LIN {X 0,Y 139.124,Z 614.225,A -85,B 0,C 180,E1 -24904.524,E2 -24904.524} C_VEL
LIN {X 0,Y 138.778,Z 622.355,A -85,B 0,C 180,E1 -24907.678,E2 -24907.678} C_VEL
LIN {X 0,Y 138.183,Z 627.369,A -85,B 0,C 180,E1 -24909.922,E2 -24909.922} C_VEL
LIN {X 0,Y 136.601,Z 635.445,A -85,B 0,C 180,E1 -24914.33,E2 -24914.33} C_VEL
LIN {X 0,Y 136.009,Z 642.268,A -85,B 0,C 180,E1 -24919.047,E2 -24919.047} C_VEL
LIN {X 0,Y 136.236,Z 647.891,A -85,B 0,C 180,E1 -24924.078,E2 -24924.078} C_VEL
LIN {X 0,Y 136.959,Z 651.569,A -85,B 0,C 180,E1 -24928.53,E2 -24928.53} C_VEL
LIN {X 0,Y 137.272,Z 652.511,A -85,B 0,C 180,E1 -24930,E2 -24930} C_VEL
LIN {X 0,Y 136.446,Z 653.751,A -85,B 0,C 180,E1 -24932.953,E2 -24932.953} C_VEL
LIN {X 0,Y 135.241,Z 654.945,A -85,B 0,C 180,E1 -24939.122,E2 -24939.122} C_VEL
LIN {X 0,Y 135.535,Z 654.719,A -85,B 0,C 180,E1 -24945.027,E2 -24945.027} C_VEL
LIN {X 0,Y 137.465,Z 653.171,A -85,B 0,C 180,E1 -24950.971,E2 -24950.971} C_VEL
LIN {X 0,Y 141.156,Z 650.311,A -85,B 0,C 180,E1 -24956.622,E2 -24956.622} C_VEL
LIN {X 0,Y 146.54,Z 646.045,A -85,B 0,C 180,E1 -24961.841,E2 -24961.841} C_VEL
LIN {X 0,Y 151.131,Z 641.889,A -85,B 0,C 180,E1 -24965.542,E2 -24965.542} C_VEL
LIN {X 0,Y 157.922,Z 634.932,A -85,B 0,C 180,E1 -24970.188,E2 -24970.188} C_VEL
LIN {X 0,Y 163.15,Z 628.696,A -85,B 0,C 180,E1 -24973.57,E2 -24973.57} C_VEL
LIN {X 0,Y 169.127,Z 620.28,A -85,B 0,C 180,E1 -24977.528,E2 -24977.528} C_VEL
LIN {X 0,Y 174.471,Z 611.295,A -85,B 0,C 180,E1 -24981.463,E2 -24981.463} C_VEL
LIN {X 0,Y 175.351,Z 609.732,A -85,B 0,C 180,E1 -24982.142,E2 -24982.142} C_VEL
LIN {X 0,Y 176.005,Z 607.9,A -85,B 0,C 180,E1 -24983.205,E2 -24983.205} C_VEL
LIN {X 0,Y 176.463,Z 604.236,A -85,B 0,C 180,E1 -24986.112,E2 -24986.112} C_VEL
LIN {X 0,Y 176.98,Z 601.228,A -85,B 0,C 180,E1 -24988.92,E2 -24988.92} C_VEL
LIN {X 0,Y 177.146,Z 597.841,A -85,B 0,C 180,E1 -24994.126,E2 -24994.126} C_VEL
LIN {X 0,Y 177.528,Z 596.674,A -85,B 0,C 180,E1 -24996.68,E2 -24996.68} C_VEL
LIN {X 0,Y 177.92,Z 595.956,A -85,B 0,C 180,E1 -24999.176,E2 -24999.176} C_VEL
LIN {X 0,Y 178.33,Z 595.956,A -85,B 0,C 180,E1 -25002.881,E2 -25002.881} C_VEL
LIN {X 0,Y 178.144,Z 596.469,A -85,B 0,C 180,E1 -25004.127,E2 -25004.127} C_VEL
LIN {X 0,Y 176.937,Z 598.219,A -85,B 0,C 180,E1 -25005.914,E2 -25005.914} C_VEL
LIN {X 0,Y 173.626,Z 602.149,A -85,B 0,C 180,E1 -25008.757,E2 -25008.757} C_VEL
LIN {X 0,Y 170.434,Z 605.82,A -85,B 0,C 180,E1 -25011.758,E2 -25011.758} C_VEL
LIN {X 0,Y 170.01,Z 606.402,A -85,B 0,C 180,E1 -25012.401,E2 -25012.401} C_VEL
LIN {X 0,Y 168.927,Z 607.829,A -85,B 0,C 180,E1 -25014.03,E2 -25014.03} C_VEL
LIN {X 0,Y 161.536,Z 613.41,A -85,B 0,C 180,E1 -25017.507,E2 -25017.507} C_VEL
LIN {X 0,Y 154.657,Z 617.635,A -85,B 0,C 180,E1 -25021.293,E2 -25021.293} C_VEL
LIN {X 0,Y 148.282,Z 620.597,A -85,B 0,C 180,E1 -25025.54,E2 -25025.54} C_VEL
LIN {X 0,Y 142.787,Z 622.288,A -85,B 0,C 180,E1 -25030.13,E2 -25030.13} C_VEL
LIN {X 0,Y 138.192,Z 622.79,A -85,B 0,C 180,E1 -25034.919,E2 -25034.919} C_VEL
LIN {X 0,Y 134.595,Z 622.122,A -85,B 0,C 180,E1 -25039.965,E2 -25039.965} C_VEL
LIN {X 0,Y 131.938,Z 620.292,A -85,B 0,C 180,E1 -25045.224,E2 -25045.224} C_VEL
LIN {X 0,Y 130.327,Z 617.426,A -85,B 0,C 180,E1 -25050.364,E2 -25050.364} C_VEL
LIN {X 0,Y 129.639,Z 613.408,A -85,B 0,C 180,E1 -25055.591,E2 -25055.591} C_VEL
LIN {X 0,Y 129.857,Z 607.36,A -85,B 0,C 180,E1 -25061.527,E2 -25061.527} C_VEL
LIN {X 0,Y 131.057,Z 600.193,A -85,B 0,C 180,E1 -25066.903,E2 -25066.903} C_VEL
LIN {X 0,Y 132.845,Z 591.924,A -85,B 0,C 180,E1 -25071.769,E2 -25071.769} C_VEL
LIN {X 0,Y 134.732,Z 584.083,A -85,B 0,C 180,E1 -25075.486,E2 -25075.486} C_VEL
LIN {X 0,Y 137.374,Z 573.433,A -85,B 0,C 180,E1 -25079.54,E2 -25079.54} C_VEL
LIN {X 0,Y 139.043,Z 566.504,A -85,B 0,C 180,E1 -25081.714,E2 -25081.714} C_VEL
LIN {X 0,Y 136.816,Z 556.881,A -85,B 0,C 180,E1 -25084.925,E2 -25084.925} C_VEL
LIN {X 0,Y 133.873,Z 546.539,A -85,B 0,C 180,E1 -25088.034,E2 -25088.034} C_VEL
LIN {X 0,Y 130.098,Z 535.182,A -85,B 0,C 180,E1 -25091.087,E2 -25091.087} C_VEL
LIN {X 0,Y 129.19,Z 532.394,A -85,B 0,C 180,E1 -25091.874,E2 -25091.874} C_VEL
LIN {X 0,Y 129.373,Z 532.372,A -85,B 0,C 180,E1 -25097.917,E2 -25097.917} C_VEL
LIN {X 0,Y 129.478,Z 532.358,A -85,B 0,C 180,E1 -25100.628,E2 -25100.628} C_VEL
LIN {X 0,Y 130.088,Z 532.28,A -85,B 0,C 180,E1 -25110,E2 -25110} C_VEL
LIN {X 0,Y 129.466,Z 532.353,A -85,B 0,C 180,E1 -25119.372,E2 -25119.372} C_VEL
LIN {X 0,Y 129.308,Z 532.377,A -85,B 0,C 180,E1 -25122.556,E2 -25122.556} C_VEL
LIN {X 0,Y 129.152,Z 532.394,A -85,B 0,C 180,E1 -25129.056,E2 -25129.056} C_VEL
LIN {X 0,Y 129.11,Z 532.402,A -85,B 0,C 180,E1 -25132.398,E2 -25132.398} C_VEL
LIN {X 0,Y 129.019,Z 532.415,A -85,B 0,C 180,E1 -25139.357,E2 -25139.357} C_VEL
LIN {X 0,Y 128.958,Z 532.416,A -85,B 0,C 180,E1 -25145.165,E2 -25145.165} C_VEL
LIN {X 0,Y 128.924,Z 532.424,A -85,B 0,C 180,E1 -25150.855,E2 -25150.855} C_VEL
LIN {X 0,Y 128.913,Z 532.425,A -85,B 0,C 180,E1 -25155.131,E2 -25155.131} C_VEL
LIN {X 0,Y 128.937,Z 532.42,A -85,B 0,C 180,E1 -25159.738,E2 -25159.738} C_VEL
LIN {X 0,Y 128.982,Z 532.418,A -85,B 0,C 180,E1 -25164.817,E2 -25164.817} C_VEL
LIN {X 0,Y 129.053,Z 532.403,A -85,B 0,C 180,E1 -25170.65,E2 -25170.65} C_VEL
LIN {X 0,Y 129.108,Z 532.397,A -85,B 0,C 180,E1 -25177.727,E2 -25177.727} C_VEL
LIN {X 0,Y 129.154,Z 532.395,A -85,B 0,C 180,E1 -25180.943,E2 -25180.943} C_VEL
LIN {X 0,Y 129.391,Z 532.362,A -85,B 0,C 180,E1 -25187.874,E2 -25187.874} C_VEL
LIN {X 0,Y 129.474,Z 532.357,A -85,B 0,C 180,E1 -25190.627,E2 -25190.627} C_VEL
LIN {X 0,Y 130.084,Z 532.28,A -85,B 0,C 180,E1 -25199.999,E2 -25199.999} C_VEL
LIN {X 0,Y 129.47,Z 532.357,A -85,B 0,C 180,E1 -25209.372,E2 -25209.372} C_VEL
LIN {X 0,Y 129.178,Z 532.393,A -85,B 0,C 180,E1 -25215.784,E2 -25215.784} C_VEL
LIN {X 0,Y 129.148,Z 532.396,A -85,B 0,C 180,E1 -25219.056,E2 -25219.056} C_VEL
LIN {X 0,Y 129.107,Z 532.397,A -85,B 0,C 180,E1 -25222.398,E2 -25222.398} C_VEL
LIN {X 0,Y 129.061,Z 532.404,A -85,B 0,C 180,E1 -25229.393,E2 -25229.393} C_VEL
LIN {X 0,Y 129.162,Z 532.55,A -85,B 0,C 180,E1 -25231.351,E2 -25231.351} C_VEL
LIN {X 0,Y 130.037,Z 536.916,A -85,B 0,C 180,E1 -25236.477,E2 -25236.477} C_VEL
LIN {X 0,Y 131.181,Z 542.343,A -85,B 0,C 180,E1 -25242.498,E2 -25242.498} C_VEL
LIN {X 0,Y 132.35,Z 547.595,A -85,B 0,C 180,E1 -25248.023,E2 -25248.023} C_VEL
LIN {X 0,Y 132.432,Z 549.569,A -85,B 0,C 180,E1 -25250.036,E2 -25250.036} C_VEL
LIN {X 0,Y 132.944,Z 563.477,A -85,B 0,C 180,E1 -25251.783,E2 -25251.783} C_VEL
LIN {X 0,Y 133.092,Z 576.046,A -85,B 0,C 180,E1 -25253.881,E2 -25253.881} C_VEL
LIN {X 0,Y 132.946,Z 588.199,A -85,B 0,C 180,E1 -25256.467,E2 -25256.467} C_VEL
LIN {X 0,Y 132.625,Z 600.647,A -85,B 0,C 180,E1 -25259.774,E2 -25259.774} C_VEL
LIN {X 0,Y 132.148,Z 612.046,A -85,B 0,C 180,E1 -25263.551,E2 -25263.551} C_VEL
LIN {X 0,Y 131.728,Z 621.194,A -85,B 0,C 180,E1 -25267.244,E2 -25267.244} C_VEL
LIN {X 0,Y 131.213,Z 626.26,A -85,B 0,C 180,E1 -25269.626,E2 -25269.626} C_VEL
LIN {X 0,Y 129.594,Z 634.342,A -85,B 0,C 180,E1 -25274.267,E2 -25274.267} C_VEL
LIN {X 0,Y 129.068,Z 640.329,A -85,B 0,C 180,E1 -25278.558,E2 -25278.558} C_VEL
LIN {X 0,Y 129.218,Z 646.012,A -85,B 0,C 180,E1 -25283.756,E2 -25283.756} C_VEL
LIN {X 0,Y 129.958,Z 649.876,A -85,B 0,C 180,E1 -25288.451,E2 -25288.451} C_VEL
LIN {X 0,Y 130.272,Z 650.893,A -85,B 0,C 180,E1 -25290,E2 -25290} C_VEL
LIN {X 0,Y 129.457,Z 652.211,A -85,B 0,C 180,E1 -25293.112,E2 -25293.112} C_VEL
LIN {X 0,Y 128.248,Z 653.603,A -85,B 0,C 180,E1 -25299.463,E2 -25299.463} C_VEL
LIN {X 0,Y 128.654,Z 653.596,A -85,B 0,C 180,E1 -25305.851,E2 -25305.851} C_VEL
LIN {X 0,Y 130.819,Z 652.241,A -85,B 0,C 180,E1 -25312.091,E2 -25312.091} C_VEL
LIN {X 0,Y 134.819,Z 649.603,A -85,B 0,C 180,E1 -25317.981,E2 -25317.981} C_VEL
LIN {X 0,Y 140.512,Z 645.643,A -85,B 0,C 180,E1 -25323.381,E2 -25323.381} C_VEL
LIN {X 0,Y 145.336,Z 641.669,A -85,B 0,C 180,E1 -25327.191,E2 -25327.191} C_VEL
LIN {X 0,Y 152.521,Z 635.126,A -85,B 0,C 180,E1 -25331.925,E2 -25331.925} C_VEL
LIN {X 0,Y 158.93,Z 628.094,A -85,B 0,C 180,E1 -25335.939,E2 -25335.939} C_VEL
LIN {X 0,Y 164.332,Z 621.22,A -85,B 0,C 180,E1 -25339.387,E2 -25339.387} C_VEL
LIN {X 0,Y 169.825,Z 613.116,A -85,B 0,C 180,E1 -25343.203,E2 -25343.203} C_VEL
LIN {X 0,Y 170.334,Z 612.196,A -85,B 0,C 180,E1 -25343.71,E2 -25343.71} C_VEL
LIN {X 0,Y 170.885,Z 610.061,A -85,B 0,C 180,E1 -25345.341,E2 -25345.341} C_VEL
LIN {X 0,Y 171.754,Z 605.979,A -85,B 0,C 180,E1 -25349.239,E2 -25349.239} C_VEL
LIN {X 0,Y 172.018,Z 602.978,A -85,B 0,C 180,E1 -25354.007,E2 -25354.007} C_VEL
LIN {X 0,Y 172.318,Z 601.996,A -85,B 0,C 180,E1 -25355.931,E2 -25355.931} C_VEL
LIN {X 0,Y 172.837,Z 600.906,A -85,B 0,C 180,E1 -25359.269,E2 -25359.269} C_VEL
LIN {X 0,Y 173.224,Z 600.854,A -85,B 0,C 180,E1 -25363.501,E2 -25363.501} C_VEL
LIN {X 0,Y 172.812,Z 601.76,A -85,B 0,C 180,E1 -25365.877,E2 -25365.877} C_VEL
LIN {X 0,Y 171.016,Z 604.884,A -85,B 0,C 180,E1 -25370.539,E2 -25370.539} C_VEL
LIN {X 0,Y 170.01,Z 606.402,A -85,B 0,C 180,E1 -25372.401,E2 -25372.401} C_VEL
LIN {X 0,Y 168.774,Z 607.616,A -85,B 0,C 180,E1 -25373.298,E2 -25373.298} C_VEL
LIN {X 0,Y 165.714,Z 609.887,A -85,B 0,C 180,E1 -25374.189,E2 -25374.189} C_VEL
LIN {X 0,Y 157.995,Z 614.59,A -85,B 0,C 180,E1 -25375.568,E2 -25375.568} C_VEL
LIN {X 0,Y 155.144,Z 616.213,A -85,B 0,C 180,E1 -25376.521,E2 -25376.521} C_VEL
LIN {X 0,Y 147.6,Z 620.166,A -85,B 0,C 180,E1 -25380.681,E2 -25380.681} C_VEL
LIN {X 0,Y 141.114,Z 622.614,A -85,B 0,C 180,E1 -25385.07,E2 -25385.07} C_VEL
LIN {X 0,Y 135.514,Z 623.818,A -85,B 0,C 180,E1 -25389.806,E2 -25389.806} C_VEL
LIN {X 0,Y 130.246,Z 623.781,A -85,B 0,C 180,E1 -25395.653,E2 -25395.653} C_VEL
LIN {X 0,Y 127.228,Z 622.785,A -85,B 0,C 180,E1 -25400.102,E2 -25400.102} C_VEL
LIN {X 0,Y 124.644,Z 620.591,A -85,B 0,C 180,E1 -25405.556,E2 -25405.556} C_VEL
LIN {X 0,Y 123.1,Z 617.313,A -85,B 0,C 180,E1 -25411.086,E2 -25411.086} C_VEL
LIN {X 0,Y 122.515,Z 612.937,A -85,B 0,C 180,E1 -25416.571,E2 -25416.571} C_VEL
LIN {X 0,Y 122.82,Z 607.4,A -85,B 0,C 180,E1 -25421.936,E2 -25421.936} C_VEL
LIN {X 0,Y 124.068,Z 600.212,A -85,B 0,C 180,E1 -25427.427,E2 -25427.427} C_VEL
LIN {X 0,Y 125.769,Z 592.618,A -85,B 0,C 180,E1 -25432.07,E2 -25432.07} C_VEL
LIN {X 0,Y 128.139,Z 583.04,A -85,B 0,C 180,E1 -25436.738,E2 -25436.738} C_VEL
LIN {X 0,Y 130.997,Z 572.004,A -85,B 0,C 180,E1 -25440.958,E2 -25440.958} C_VEL
LIN {X 0,Y 131.998,Z 568.011,A -85,B 0,C 180,E1 -25442.232,E2 -25442.232} C_VEL
LIN {X 0,Y 131.502,Z 564.714,A -85,B 0,C 180,E1 -25443.41,E2 -25443.41} C_VEL
LIN {X 0,Y 128.765,Z 553.774,A -85,B 0,C 180,E1 -25447.114,E2 -25447.114} C_VEL
LIN {X 0,Y 125.494,Z 543.105,A -85,B 0,C 180,E1 -25450.365,E2 -25450.365} C_VEL
LIN {X 0,Y 122.16,Z 533.27,A -85,B 0,C 180,E1 -25453.174,E2 -25453.174} C_VEL
LIN {X 0,Y 122.409,Z 533.238,A -85,B 0,C 180,E1 -25460.081,E2 -25460.081} C_VEL
LIN {X 0,Y 122.598,Z 533.214,A -85,B 0,C 180,E1 -25466.713,E2 -25466.713} C_VEL
LIN {X 0,Y 123.041,Z 533.158,A -85,B 0,C 180,E1 -25470,E2 -25470} C_VEL
LIN {X 0,Y 122.417,Z 533.234,A -85,B 0,C 180,E1 -25476.593,E2 -25476.593} C_VEL
LIN {X 0,Y 122.294,Z 533.251,A -85,B 0,C 180,E1 -25482.318,E2 -25482.318} C_VEL
LIN {X 0,Y 122.106,Z 533.269,A -85,B 0,C 180,E1 -25486.725,E2 -25486.725} C_VEL
LIN {X 0,Y 122.03,Z 533.285,A -85,B 0,C 180,E1 -25492.854,E2 -25492.854} C_VEL
LIN {X 0,Y 121.941,Z 533.292,A -85,B 0,C 180,E1 -25497.456,E2 -25497.456} C_VEL
LIN {X 0,Y 121.9,Z 533.3,A -85,B 0,C 180,E1 -25501.257,E2 -25501.257} C_VEL
LIN {X 0,Y 121.883,Z 533.299,A -85,B 0,C 180,E1 -25506.168,E2 -25506.168} C_VEL
LIN {X 0,Y 121.865,Z 533.301,A -85,B 0,C 180,E1 -25511.432,E2 -25511.432} C_VEL
LIN {X 0,Y 121.866,Z 533.304,A -85,B 0,C 180,E1 -25518.565,E2 -25518.565} C_VEL
LIN {X 0,Y 121.934,Z 533.296,A -85,B 0,C 180,E1 -25524.803,E2 -25524.803} C_VEL
LIN {X 0,Y 121.943,Z 533.287,A -85,B 0,C 180,E1 -25529.826,E2 -25529.826} C_VEL
LIN {X 0,Y 121.984,Z 533.289,A -85,B 0,C 180,E1 -25536.214,E2 -25536.214} C_VEL
LIN {X 0,Y 122.046,Z 533.278,A -85,B 0,C 180,E1 -25539.786,E2 -25539.786} C_VEL
LIN {X 0,Y 122.24,Z 533.252,A -85,B 0,C 180,E1 -25546.704,E2 -25546.704} C_VEL
LIN {X 0,Y 122.41,Z 533.235,A -85,B 0,C 180,E1 -25550.081,E2 -25550.081} C_VEL
LIN {X 0,Y 122.593,Z 533.208,A -85,B 0,C 180,E1 -25556.713,E2 -25556.713} C_VEL
LIN {X 0,Y 123.038,Z 533.158,A -85,B 0,C 180,E1 -25559.999,E2 -25559.999} C_VEL
LIN {X 0,Y 122.415,Z 533.234,A -85,B 0,C 180,E1 -25566.593,E2 -25566.593} C_VEL
LIN {X 0,Y 122.397,Z 533.237,A -85,B 0,C 180,E1 -25569.918,E2 -25569.918} C_VEL
LIN {X 0,Y 122.097,Z 533.276,A -85,B 0,C 180,E1 -25576.726,E2 -25576.726} C_VEL
LIN {X 0,Y 122.022,Z 533.281,A -85,B 0,C 180,E1 -25582.848,E2 -25582.848} C_VEL
LIN {X 0,Y 122.107,Z 533.333,A -85,B 0,C 180,E1 -25590.877,E2 -25590.877} C_VEL
LIN {X 0,Y 123.083,Z 538.211,A -85,B 0,C 180,E1 -25596.928,E2 -25596.928} C_VEL
LIN {X 0,Y 124.168,Z 543.249,A -85,B 0,C 180,E1 -25602.781,E2 -25602.781} C_VEL
LIN {X 0,Y 125.324,Z 548.529,A -85,B 0,C 180,E1 -25608.622,E2 -25608.622} C_VEL
LIN {X 0,Y 126.051,Z 554.121,A -85,B 0,C 180,E1 -25609.391,E2 -25609.391} C_VEL
LIN {X 0,Y 126.244,Z 567.958,A -85,B 0,C 180,E1 -25611.465,E2 -25611.465} C_VEL
LIN {X 0,Y 126.188,Z 580.638,A -85,B 0,C 180,E1 -25613.965,E2 -25613.965} C_VEL
LIN {X 0,Y 125.809,Z 593.441,A -85,B 0,C 180,E1 -25617.168,E2 -25617.168} C_VEL
LIN {X 0,Y 125.369,Z 604.623,A -85,B 0,C 180,E1 -25620.626,E2 -25620.626} C_VEL
LIN {X 0,Y 124.946,Z 614.655,A -85,B 0,C 180,E1 -25624.431,E2 -25624.431} C_VEL
LIN {X 0,Y 124.464,Z 623.437,A -85,B 0,C 180,E1 -25628.468,E2 -25628.468} C_VEL
LIN {X 0,Y 123.003,Z 630.608,A -85,B 0,C 180,E1 -25632.545,E2 -25632.545} C_VEL
LIN {X 0,Y 122.147,Z 638.257,A -85,B 0,C 180,E1 -25637.993,E2 -25637.993} C_VEL
LIN {X 0,Y 122.21,Z 644.067,A -85,B 0,C 180,E1 -25643.396,E2 -25643.396} C_VEL
LIN {X 0,Y 122.953,Z 648.144,A -85,B 0,C 180,E1 -25648.363,E2 -25648.363} C_VEL
LIN {X 0,Y 123.273,Z 649.244,A -85,B 0,C 180,E1 -25650,E2 -25650} C_VEL
LIN {X 0,Y 122.455,Z 650.667,A -85,B 0,C 180,E1 -25653.291,E2 -25653.291} C_VEL
LIN {X 0,Y 121.267,Z 652.206,A -85,B 0,C 180,E1 -25660.013,E2 -25660.013} C_VEL
LIN {X 0,Y 121.811,Z 652.395,A -85,B 0,C 180,E1 -25666.767,E2 -25666.767} C_VEL
LIN {X 0,Y 124.233,Z 651.296,A -85,B 0,C 180,E1 -25673.329,E2 -25673.329} C_VEL
LIN {X 0,Y 128.558,Z 648.898,A -85,B 0,C 180,E1 -25679.473,E2 -25679.473} C_VEL
LIN {X 0,Y 134.608,Z 645.172,A -85,B 0,C 180,E1 -25685.053,E2 -25685.053} C_VEL
LIN {X 0,Y 141.489,Z 640.048,A -85,B 0,C 180,E1 -25690.221,E2 -25690.221} C_VEL
LIN {X 0,Y 147.25,Z 635.214,A -85,B 0,C 180,E1 -25693.794,E2 -25693.794} C_VEL
LIN {X 0,Y 153.976,Z 628.592,A -85,B 0,C 180,E1 -25697.878,E2 -25697.878} C_VEL
LIN {X 0,Y 159.664,Z 622.069,A -85,B 0,C 180,E1 -25701.382,E2 -25701.382} C_VEL
LIN {X 0,Y 164.294,Z 616.161,A -85,B 0,C 180,E1 -25704.368,E2 -25704.368} C_VEL
LIN {X 0,Y 164.978,Z 614.895,A -85,B 0,C 180,E1 -25705.219,E2 -25705.219} C_VEL
LIN {X 0,Y 166.253,Z 610.512,A -85,B 0,C 180,E1 -25709.518,E2 -25709.518} C_VEL
LIN {X 0,Y 166.781,Z 607.186,A -85,B 0,C 180,E1 -25715.078,E2 -25715.078} C_VEL
LIN {X 0,Y 167.218,Z 606.107,A -85,B 0,C 180,E1 -25717.775,E2 -25717.775} C_VEL
LIN {X 0,Y 167.563,Z 605.463,A -85,B 0,C 180,E1 -25720.395,E2 -25720.395} C_VEL
LIN {X 0,Y 167.735,Z 605.424,A -85,B 0,C 180,E1 -25722.945,E2 -25722.945} C_VEL
LIN {X 0,Y 167.301,Z 606.032,A -85,B 0,C 180,E1 -25725.402,E2 -25725.402} C_VEL
LIN {X 0,Y 166.263,Z 607.365,A -85,B 0,C 180,E1 -25727.799,E2 -25727.799} C_VEL
LIN {X 0,Y 165.126,Z 608.814,A -85,B 0,C 180,E1 -25730.198,E2 -25730.198} C_VEL
LIN {X 0,Y 163.561,Z 610.602,A -85,B 0,C 180,E1 -25732.594,E2 -25732.594} C_VEL
LIN {X 0,Y 155.144,Z 616.213,A -85,B 0,C 180,E1 -25736.521,E2 -25736.521} C_VEL
LIN {X 0,Y 151.396,Z 618.235,A -85,B 0,C 180,E1 -25738.058,E2 -25738.058} C_VEL
LIN {X 0,Y 144.069,Z 621.349,A -85,B 0,C 180,E1 -25740.35,E2 -25740.35} C_VEL
LIN {X 0,Y 136.878,Z 623.722,A -85,B 0,C 180,E1 -25742.936,E2 -25742.936} C_VEL
LIN {X 0,Y 133.446,Z 624.538,A -85,B 0,C 180,E1 -25744.93,E2 -25744.93} C_VEL
LIN {X 0,Y 128.225,Z 625.196,A -85,B 0,C 180,E1 -25749.465,E2 -25749.465} C_VEL
LIN {X 0,Y 123.531,Z 624.802,A -85,B 0,C 180,E1 -25754.717,E2 -25754.717} C_VEL
LIN {X 0,Y 119.671,Z 623.168,A -85,B 0,C 180,E1 -25760.633,E2 -25760.633} C_VEL
LIN {X 0,Y 117.305,Z 620.71,A -85,B 0,C 180,E1 -25766.013,E2 -25766.013} C_VEL
LIN {X 0,Y 115.867,Z 617.011,A -85,B 0,C 180,E1 -25771.876,E2 -25771.876} C_VEL
LIN {X 0,Y 115.427,Z 612.238,A -85,B 0,C 180,E1 -25777.67,E2 -25777.67} C_VEL
LIN {X 0,Y 115.941,Z 606.327,A -85,B 0,C 180,E1 -25783.33,E2 -25783.33} C_VEL
LIN {X 0,Y 117.322,Z 599.084,A -85,B 0,C 180,E1 -25788.78,E2 -25788.78} C_VEL
LIN {X 0,Y 119.372,Z 590.5,A -85,B 0,C 180,E1 -25793.931,E2 -25793.931} C_VEL
LIN {X 0,Y 121.568,Z 582.032,A -85,B 0,C 180,E1 -25798.023,E2 -25798.023} C_VEL
LIN {X 0,Y 124.265,Z 571.835,A -85,B 0,C 180,E1 -25801.98,E2 -25801.98} C_VEL
LIN {X 0,Y 125.052,Z 568.008,A -85,B 0,C 180,E1 -25803.281,E2 -25803.281} C_VEL
LIN {X 0,Y 122.764,Z 558.461,A -85,B 0,C 180,E1 -25806.822,E2 -25806.822} C_VEL
LIN {X 0,Y 119.839,Z 548.155,A -85,B 0,C 180,E1 -25810.293,E2 -25810.293} C_VEL
LIN {X 0,Y 116.565,Z 538.35,A -85,B 0,C 180,E1 -25813.357,E2 -25813.357} C_VEL
LIN {X 0,Y 115.104,Z 534.149,A -85,B 0,C 180,E1 -25814.619,E2 -25814.619} C_VEL
LIN {X 0,Y 115.325,Z 534.121,A -85,B 0,C 180,E1 -25819.465,E2 -25819.465} C_VEL
LIN {X 0,Y 115.522,Z 534.095,A -85,B 0,C 180,E1 -25826.512,E2 -25826.512} C_VEL
LIN {X 0,Y 115.993,Z 534.036,A -85,B 0,C 180,E1 -25830,E2 -25830} C_VEL
LIN {X 0,Y 115.358,Z 534.112,A -85,B 0,C 180,E1 -25836.998,E2 -25836.998} C_VEL
LIN {X 0,Y 115.237,Z 534.13,A -85,B 0,C 180,E1 -25842.626,E2 -25842.626} C_VEL
LIN {X 0,Y 115.01,Z 534.153,A -85,B 0,C 180,E1 -25847.79,E2 -25847.79} C_VEL
LIN {X 0,Y 114.949,Z 534.164,A -85,B 0,C 180,E1 -25853.49,E2 -25853.49} C_VEL
LIN {X 0,Y 114.857,Z 534.178,A -85,B 0,C 180,E1 -25861.055,E2 -25861.055} C_VEL
LIN {X 0,Y 114.777,Z 534.188,A -85,B 0,C 180,E1 -25867.757,E2 -25867.757} C_VEL
LIN {X 0,Y 114.779,Z 534.181,A -85,B 0,C 180,E1 -25872.711,E2 -25872.711} C_VEL
LIN {X 0,Y 114.788,Z 534.186,A -85,B 0,C 180,E1 -25877.662,E2 -25877.662} C_VEL
LIN {X 0,Y 114.797,Z 534.18,A -85,B 0,C 180,E1 -25882.737,E2 -25882.737} C_VEL
LIN {X 0,Y 114.869,Z 534.171,A -85,B 0,C 180,E1 -25888.932,E2 -25888.932} C_VEL
LIN {X 0,Y 114.947,Z 534.165,A -85,B 0,C 180,E1 -25896.508,E2 -25896.508} C_VEL
LIN {X 0,Y 115.012,Z 534.158,A -85,B 0,C 180,E1 -25902.209,E2 -25902.209} C_VEL
LIN {X 0,Y 115.25,Z 534.122,A -85,B 0,C 180,E1 -25907.339,E2 -25907.339} C_VEL
LIN {X 0,Y 115.363,Z 534.114,A -85,B 0,C 180,E1 -25913.001,E2 -25913.001} C_VEL
LIN {X 0,Y 115.989,Z 534.036,A -85,B 0,C 180,E1 -25919.999,E2 -25919.999} C_VEL
LIN {X 0,Y 115.356,Z 534.115,A -85,B 0,C 180,E1 -25926.998,E2 -25926.998} C_VEL
LIN {X 0,Y 115.208,Z 534.128,A -85,B 0,C 180,E1 -25932.567,E2 -25932.567} C_VEL
LIN {X 0,Y 115.004,Z 534.159,A -85,B 0,C 180,E1 -25937.791,E2 -25937.791} C_VEL
LIN {X 0,Y 114.944,Z 534.165,A -85,B 0,C 180,E1 -25943.489,E2 -25943.489} C_VEL
LIN {X 0,Y 115.039,Z 534.26,A -85,B 0,C 180,E1 -25950.602,E2 -25950.602} C_VEL
LIN {X 0,Y 115.779,Z 537.749,A -85,B 0,C 180,E1 -25955.216,E2 -25955.216} C_VEL
LIN {X 0,Y 116.821,Z 542.751,A -85,B 0,C 180,E1 -25961.434,E2 -25961.434} C_VEL
LIN {X 0,Y 117.901,Z 547.405,A -85,B 0,C 180,E1 -25966.963,E2 -25966.963} C_VEL
LIN {X 0,Y 119.401,Z 553.61,A -85,B 0,C 180,E1 -25968.035,E2 -25968.035} C_VEL
LIN {X 0,Y 119.524,Z 566.395,A -85,B 0,C 180,E1 -25970.065,E2 -25970.065} C_VEL
LIN {X 0,Y 119.356,Z 579.884,A -85,B 0,C 180,E1 -25972.876,E2 -25972.876} C_VEL
LIN {X 0,Y 118.936,Z 592.084,A -85,B 0,C 180,E1 -25976.11,E2 -25976.11} C_VEL
LIN {X 0,Y 118.412,Z 603.124,A -85,B 0,C 180,E1 -25979.703,E2 -25979.703} C_VEL
LIN {X 0,Y 117.976,Z 612.321,A -85,B 0,C 180,E1 -25983.324,E2 -25983.324} C_VEL
LIN {X 0,Y 117.575,Z 620.439,A -85,B 0,C 180,E1 -25987.137,E2 -25987.137} C_VEL
LIN {X 0,Y 116.979,Z 625.275,A -85,B 0,C 180,E1 -25989.791,E2 -25989.791} C_VEL
LIN {X 0,Y 115.438,Z 633.097,A -85,B 0,C 180,E1 -25995.005,E2 -25995.005} C_VEL
LIN {X 0,Y 115.112,Z 638.487,A -85,B 0,C 180,E1 -25999.446,E2 -25999.446} C_VEL
LIN {X 0,Y 115.409,Z 643.649,A -85,B 0,C 180,E1 -26004.759,E2 -26004.759} C_VEL
LIN {X 0,Y 116.298,Z 647.516,A -85,B 0,C 180,E1 -26010,E2 -26010} C_VEL
LIN {X 0,Y 115.475,Z 649.039,A -85,B 0,C 180,E1 -26013.49,E2 -26013.49} C_VEL
LIN {X 0,Y 114.312,Z 650.801,A -85,B 0,C 180,E1 -26020.629,E2 -26020.629} C_VEL
LIN {X 0,Y 115.011,Z 651.173,A -85,B 0,C 180,E1 -26027.791,E2 -26027.791} C_VEL
LIN {X 0,Y 117.716,Z 650.279,A -85,B 0,C 180,E1 -26034.704,E2 -26034.704} C_VEL
LIN {X 0,Y 122.417,Z 648.139,A -85,B 0,C 180,E1 -26041.111,E2 -26041.111} C_VEL
LIN {X 0,Y 128.834,Z 644.727,A -85,B 0,C 180,E1 -26046.875,E2 -26046.875} C_VEL
LIN {X 0,Y 136.087,Z 639.872,A -85,B 0,C 180,E1 -26052.173,E2 -26052.173} C_VEL
LIN {X 0,Y 144.003,Z 633.78,A -85,B 0,C 180,E1 -26056.902,E2 -26056.902} C_VEL
LIN {X 0,Y 151.231,Z 627.069,A -85,B 0,C 180,E1 -26061.116,E2 -26061.116} C_VEL
LIN {X 0,Y 156.512,Z 621.485,A -85,B 0,C 180,E1 -26064.286,E2 -26064.286} C_VEL
LIN {X 0,Y 159.063,Z 618.475,A -85,B 0,C 180,E1 -26065.939,E2 -26065.939} C_VEL
LIN {X 0,Y 159.989,Z 616.237,A -85,B 0,C 180,E1 -26068.188,E2 -26068.188} C_VEL
LIN {X 0,Y 160.509,Z 614.796,A -85,B 0,C 180,E1 -26069.768,E2 -26069.768} C_VEL
LIN {X 0,Y 161.005,Z 612.198,A -85,B 0,C 180,E1 -26074.119,E2 -26074.119} C_VEL
LIN {X 0,Y 161.46,Z 610.906,A -85,B 0,C 180,E1 -26076.937,E2 -26076.937} C_VEL
LIN {X 0,Y 161.857,Z 610.073,A -85,B 0,C 180,E1 -26079.674,E2 -26079.674} C_VEL
LIN {X 0,Y 162.065,Z 609.743,A -85,B 0,C 180,E1 -26082.563,E2 -26082.563} C_VEL
LIN {X 0,Y 161.642,Z 610.122,A -85,B 0,C 180,E1 -26084.879,E2 -26084.879} C_VEL
LIN {X 0,Y 160.446,Z 611.242,A -85,B 0,C 180,E1 -26087.349,E2 -26087.349} C_VEL
LIN {X 0,Y 159.047,Z 612.576,A -85,B 0,C 180,E1 -26089.82,E2 -26089.82} C_VEL
LIN {X 0,Y 158.202,Z 613.294,A -85,B 0,C 180,E1 -26090.996,E2 -26090.996} C_VEL
LIN {X 0,Y 155.394,Z 615.139,A -85,B 0,C 180,E1 -26092.416,E2 -26092.416} C_VEL
LIN {X 0,Y 147.977,Z 619.298,A -85,B 0,C 180,E1 -26095.853,E2 -26095.853} C_VEL
LIN {X 0,Y 140.562,Z 622.507,A -85,B 0,C 180,E1 -26100.001,E2 -26100.001} C_VEL
LIN {X 0,Y 133.446,Z 624.538,A -85,B 0,C 180,E1 -26104.93,E2 -26104.93} C_VEL
LIN {X 0,Y 130.128,Z 625.12,A -85,B 0,C 180,E1 -26107.043,E2 -26107.043} C_VEL
LIN {X 0,Y 123.492,Z 625.797,A -85,B 0,C 180,E1 -26110.358,E2 -26110.358} C_VEL
LIN {X 0,Y 117.276,Z 625.64,A -85,B 0,C 180,E1 -26114.022,E2 -26114.022} C_VEL
LIN {X 0,Y 114.727,Z 624.976,A -85,B 0,C 180,E1 -26116.629,E2 -26116.629} C_VEL
LIN {X 0,Y 111.628,Z 622.909,A -85,B 0,C 180,E1 -26122.196,E2 -26122.196} C_VEL
LIN {X 0,Y 109.335,Z 619.318,A -85,B 0,C 180,E1 -26128.824,E2 -26128.824} C_VEL
LIN {X 0,Y 108.37,Z 614.216,A -85,B 0,C 180,E1 -26135.71,E2 -26135.71} C_VEL
LIN {X 0,Y 108.706,Z 607.554,A -85,B 0,C 180,E1 -26142.642,E2 -26142.642} C_VEL
LIN {X 0,Y 110.082,Z 600.176,A -85,B 0,C 180,E1 -26148.606,E2 -26148.606} C_VEL
LIN {X 0,Y 112.314,Z 591.044,A -85,B 0,C 180,E1 -26154.438,E2 -26154.438} C_VEL
LIN {X 0,Y 114.784,Z 581.955,A -85,B 0,C 180,E1 -26159.006,E2 -26159.006} C_VEL
LIN {X 0,Y 117.863,Z 570.675,A -85,B 0,C 180,E1 -26163.438,E2 -26163.438} C_VEL
LIN {X 0,Y 118.127,Z 569.272,A -85,B 0,C 180,E1 -26163.947,E2 -26163.947} C_VEL
LIN {X 0,Y 115.759,Z 559.19,A -85,B 0,C 180,E1 -26167.934,E2 -26167.934} C_VEL
LIN {X 0,Y 113.152,Z 549.965,A -85,B 0,C 180,E1 -26171.257,E2 -26171.257} C_VEL
LIN {X 0,Y 110.207,Z 540.979,A -85,B 0,C 180,E1 -26174.274,E2 -26174.274} C_VEL
LIN {X 0,Y 108.135,Z 535.017,A -85,B 0,C 180,E1 -26176.215,E2 -26176.215} C_VEL
LIN {X 0,Y 108.253,Z 535.003,A -85,B 0,C 180,E1 -26178.768,E2 -26178.768} C_VEL
LIN {X 0,Y 108.446,Z 534.976,A -85,B 0,C 180,E1 -26186.284,E2 -26186.284} C_VEL
LIN {X 0,Y 108.918,Z 534.917,A -85,B 0,C 180,E1 -26190,E2 -26190} C_VEL
LIN {X 0,Y 108.296,Z 534.99,A -85,B 0,C 180,E1 -26197.457,E2 -26197.457} C_VEL
LIN {X 0,Y 108.162,Z 535.012,A -85,B 0,C 180,E1 -26202.922,E2 -26202.922} C_VEL
LIN {X 0,Y 107.904,Z 535.04,A -85,B 0,C 180,E1 -26209.005,E2 -26209.005} C_VEL
LIN {X 0,Y 107.858,Z 535.046,A -85,B 0,C 180,E1 -26214.18,E2 -26214.18} C_VEL
LIN {X 0,Y 107.781,Z 535.057,A -85,B 0,C 180,E1 -26222.037,E2 -26222.037} C_VEL
LIN {X 0,Y 107.685,Z 535.071,A -85,B 0,C 180,E1 -26228.446,E2 -26228.446} C_VEL
LIN {X 0,Y 107.671,Z 535.072,A -85,B 0,C 180,E1 -26235.889,E2 -26235.889} C_VEL
LIN {X 0,Y 107.692,Z 535.063,A -85,B 0,C 180,E1 -26241.547,E2 -26241.547} C_VEL
LIN {X 0,Y 107.806,Z 535.052,A -85,B 0,C 180,E1 -26248.564,E2 -26248.564} C_VEL
LIN {X 0,Y 107.911,Z 535.039,A -85,B 0,C 180,E1 -26256.997,E2 -26256.997} C_VEL
LIN {X 0,Y 108.031,Z 535.026,A -85,B 0,C 180,E1 -26264.916,E2 -26264.916} C_VEL
LIN {X 0,Y 108.253,Z 534.996,A -85,B 0,C 180,E1 -26268.768,E2 -26268.768} C_VEL
LIN {X 0,Y 108.442,Z 534.969,A -85,B 0,C 180,E1 -26276.283,E2 -26276.283} C_VEL
LIN {X 0,Y 108.914,Z 534.918,A -85,B 0,C 180,E1 -26279.999,E2 -26279.999} C_VEL
LIN {X 0,Y 108.295,Z 534.995,A -85,B 0,C 180,E1 -26287.457,E2 -26287.457} C_VEL
LIN {X 0,Y 108.141,Z 535.008,A -85,B 0,C 180,E1 -26292.88,E2 -26292.88} C_VEL
LIN {X 0,Y 107.898,Z 535.043,A -85,B 0,C 180,E1 -26299.006,E2 -26299.006} C_VEL
LIN {X 0,Y 107.858,Z 535.048,A -85,B 0,C 180,E1 -26304.184,E2 -26304.184} C_VEL
LIN {X 0,Y 107.975,Z 535.149,A -85,B 0,C 180,E1 -26310.293,E2 -26310.293} C_VEL
LIN {X 0,Y 108.779,Z 538.913,A -85,B 0,C 180,E1 -26315.553,E2 -26315.553} C_VEL
LIN {X 0,Y 109.894,Z 543.941,A -85,B 0,C 180,E1 -26322.182,E2 -26322.182} C_VEL
LIN {X 0,Y 110.43,Z 546.246,A -85,B 0,C 180,E1 -26325.124,E2 -26325.124} C_VEL
LIN {X 0,Y 112.823,Z 554.9,A -85,B 0,C 180,E1 -26326.878,E2 -26326.878} C_VEL
LIN {X 0,Y 112.795,Z 567.936,A -85,B 0,C 180,E1 -26329.176,E2 -26329.176} C_VEL
LIN {X 0,Y 112.443,Z 581.314,A -85,B 0,C 180,E1 -26332.27,E2 -26332.27} C_VEL
LIN {X 0,Y 111.938,Z 592.794,A -85,B 0,C 180,E1 -26335.594,E2 -26335.594} C_VEL
LIN {X 0,Y 111.327,Z 604.144,A -85,B 0,C 180,E1 -26339.667,E2 -26339.667} C_VEL
LIN {X 0,Y 110.782,Z 614.313,A -85,B 0,C 180,E1 -26344.142,E2 -26344.142} C_VEL
LIN {X 0,Y 110.265,Z 622.466,A -85,B 0,C 180,E1 -26348.501,E2 -26348.501} C_VEL
LIN {X 0,Y 108.884,Z 629.423,A -85,B 0,C 180,E1 -26353.115,E2 -26353.115} C_VEL
LIN {X 0,Y 108.187,Z 636.269,A -85,B 0,C 180,E1 -26358.762,E2 -26358.762} C_VEL
LIN {X 0,Y 108.392,Z 641.643,A -85,B 0,C 180,E1 -26364.419,E2 -26364.419} C_VEL
LIN {X 0,Y 109.314,Z 645.729,A -85,B 0,C 180,E1 -26370,E2 -26370} C_VEL
LIN {X 0,Y 108.515,Z 647.359,A -85,B 0,C 180,E1 -26373.714,E2 -26373.714} C_VEL
LIN {X 0,Y 107.372,Z 649.302,A -85,B 0,C 180,E1 -26381.325,E2 -26381.325} C_VEL
LIN {X 0,Y 108.259,Z 649.906,A -85,B 0,C 180,E1 -26388.941,E2 -26388.941} C_VEL
LIN {X 0,Y 111.279,Z 649.261,A -85,B 0,C 180,E1 -26396.238,E2 -26396.238} C_VEL
LIN {X 0,Y 116.383,Z 647.358,A -85,B 0,C 180,E1 -26402.922,E2 -26402.922} C_VEL
LIN {X 0,Y 123.187,Z 644.179,A -85,B 0,C 180,E1 -26408.871,E2 -26408.871} C_VEL
LIN {X 0,Y 130.865,Z 639.684,A -85,B 0,C 180,E1 -26414.28,E2 -26414.28} C_VEL
LIN {X 0,Y 139.34,Z 633.821,A -85,B 0,C 180,E1 -26419.163,E2 -26419.163} C_VEL
LIN {X 0,Y 145.705,Z 628.554,A -85,B 0,C 180,E1 -26422.738,E2 -26422.738} C_VEL
LIN {X 0,Y 151.983,Z 622.661,A -85,B 0,C 180,E1 -26426.343,E2 -26426.343} C_VEL
LIN {X 0,Y 153.682,Z 620.68,A -85,B 0,C 180,E1 -26427.782,E2 -26427.782} C_VEL
LIN {X 0,Y 154.532,Z 618.8,A -85,B 0,C 180,E1 -26429.983,E2 -26429.983} C_VEL
LIN {X 0,Y 155.273,Z 616.019,A -85,B 0,C 180,E1 -26434.858,E2 -26434.858} C_VEL
LIN {X 0,Y 155.894,Z 614.485,A -85,B 0,C 180,E1 -26438.86,E2 -26438.86} C_VEL
LIN {X 0,Y 156.141,Z 613.884,A -85,B 0,C 180,E1 -26441.635,E2 -26441.635} C_VEL
LIN {X 0,Y 155.831,Z 613.994,A -85,B 0,C 180,E1 -26444.301,E2 -26444.301} C_VEL
LIN {X 0,Y 154.489,Z 614.883,A -85,B 0,C 180,E1 -26446.853,E2 -26446.853} C_VEL
LIN {X 0,Y 152.862,Z 616.074,A -85,B 0,C 180,E1 -26449.403,E2 -26449.403} C_VEL
LIN {X 0,Y 151.456,Z 616.923,A -85,B 0,C 180,E1 -26450.293,E2 -26450.293} C_VEL
LIN {X 0,Y 142.362,Z 621.469,A -85,B 0,C 180,E1 -26454.334,E2 -26454.334} C_VEL
LIN {X 0,Y 133.546,Z 624.65,A -85,B 0,C 180,E1 -26459.208,E2 -26459.208} C_VEL
LIN {X 0,Y 126.798,Z 626.099,A -85,B 0,C 180,E1 -26463.891,E2 -26463.891} C_VEL
LIN {X 0,Y 120.972,Z 626.407,A -85,B 0,C 180,E1 -26469.015,E2 -26469.015} C_VEL
LIN {X 0,Y 116.178,Z 625.593,A -85,B 0,C 180,E1 -26474.555,E2 -26474.555} C_VEL
LIN {X 0,Y 114.727,Z 624.976,A -85,B 0,C 180,E1 -26476.629,E2 -26476.629} C_VEL
LIN {X 0,Y 112.395,Z 624.142,A -85,B 0,C 180,E1 -26479.335,E2 -26479.335} C_VEL
LIN {X 0,Y 107.365,Z 622.292,A -85,B 0,C 180,E1 -26483.696,E2 -26483.696} C_VEL
LIN {X 0,Y 102.972,Z 619.72,A -85,B 0,C 180,E1 -26488.341,E2 -26488.341} C_VEL
LIN {X 0,Y 101.719,Z 617.683,A -85,B 0,C 180,E1 -26491.369,E2 -26491.369} C_VEL
LIN {X 0,Y 101.27,Z 611.864,A -85,B 0,C 180,E1 -26498.653,E2 -26498.653} C_VEL
LIN {X 0,Y 102.036,Z 605.22,A -85,B 0,C 180,E1 -26505.139,E2 -26505.139} C_VEL
LIN {X 0,Y 103.915,Z 596.674,A -85,B 0,C 180,E1 -26511.684,E2 -26511.684} C_VEL
LIN {X 0,Y 106.383,Z 587.528,A -85,B 0,C 180,E1 -26517.208,E2 -26517.208} C_VEL
LIN {X 0,Y 109.336,Z 577.115,A -85,B 0,C 180,E1 -26522.112,E2 -26522.112} C_VEL
LIN {X 0,Y 111.182,Z 570.353,A -85,B 0,C 180,E1 -26524.742,E2 -26524.742} C_VEL
LIN {X 0,Y 109.13,Z 561.492,A -85,B 0,C 180,E1 -26528.492,E2 -26528.492} C_VEL
LIN {X 0,Y 106.161,Z 550.701,A -85,B 0,C 180,E1 -26532.668,E2 -26532.668} C_VEL
LIN {X 0,Y 102.404,Z 539.783,A -85,B 0,C 180,E1 -26536.662,E2 -26536.662} C_VEL
LIN {X 0,Y 101.18,Z 535.884,A -85,B 0,C 180,E1 -26538.099,E2 -26538.099} C_VEL
LIN {X 0,Y 101.243,Z 535.874,A -85,B 0,C 180,E1 -26542.019,E2 -26542.019} C_VEL
LIN {X 0,Y 101.846,Z 535.798,A -85,B 0,C 180,E1 -26549.999,E2 -26549.999} C_VEL
LIN {X 0,Y 101.234,Z 535.868,A -85,B 0,C 180,E1 -26557.981,E2 -26557.981} C_VEL
LIN {X 0,Y 101.093,Z 535.893,A -85,B 0,C 180,E1 -26563.268,E2 -26563.268} C_VEL
LIN {X 0,Y 100.817,Z 535.926,A -85,B 0,C 180,E1 -26570.398,E2 -26570.398} C_VEL
LIN {X 0,Y 100.777,Z 535.925,A -85,B 0,C 180,E1 -26574.957,E2 -26574.957} C_VEL
LIN {X 0,Y 100.69,Z 535.937,A -85,B 0,C 180,E1 -26583.112,E2 -26583.112} C_VEL
LIN {X 0,Y 100.636,Z 535.948,A -85,B 0,C 180,E1 -26589.806,E2 -26589.806} C_VEL
LIN {X 0,Y 100.642,Z 535.948,A -85,B 0,C 180,E1 -26595.706,E2 -26595.706} C_VEL
LIN {X 0,Y 100.63,Z 535.943,A -85,B 0,C 180,E1 -26601.054,E2 -26601.054} C_VEL
LIN {X 0,Y 100.698,Z 535.942,A -85,B 0,C 180,E1 -26606.878,E2 -26606.878} C_VEL
LIN {X 0,Y 100.787,Z 535.93,A -85,B 0,C 180,E1 -26615.266,E2 -26615.266} C_VEL
LIN {X 0,Y 100.816,Z 535.921,A -85,B 0,C 180,E1 -26619.6,E2 -26619.6} C_VEL
LIN {X 0,Y 101.101,Z 535.885,A -85,B 0,C 180,E1 -26626.705,E2 -26626.705} C_VEL
LIN {X 0,Y 101.241,Z 535.874,A -85,B 0,C 180,E1 -26632.018,E2 -26632.018} C_VEL
LIN {X 0,Y 101.842,Z 535.799,A -85,B 0,C 180,E1 -26639.999,E2 -26639.999} C_VEL
LIN {X 0,Y 101.231,Z 535.875,A -85,B 0,C 180,E1 -26647.98,E2 -26647.98} C_VEL
LIN {X 0,Y 101.076,Z 535.887,A -85,B 0,C 180,E1 -26653.234,E2 -26653.234} C_VEL
LIN {X 0,Y 100.812,Z 535.922,A -85,B 0,C 180,E1 -26660.399,E2 -26660.399} C_VEL
LIN {X 0,Y 100.774,Z 535.932,A -85,B 0,C 180,E1 -26664.958,E2 -26664.958} C_VEL
LIN {X 0,Y 100.929,Z 536.045,A -85,B 0,C 180,E1 -26670.031,E2 -26670.031} C_VEL
LIN {X 0,Y 101.78,Z 540.026,A -85,B 0,C 180,E1 -26675.936,E2 -26675.936} C_VEL
LIN {X 0,Y 102.62,Z 543.7,A -85,B 0,C 180,E1 -26681.12,E2 -26681.12} C_VEL
LIN {X 0,Y 102.937,Z 545.117,A -85,B 0,C 180,E1 -26683.057,E2 -26683.057} C_VEL
LIN {X 0,Y 104.156,Z 549.108,A -85,B 0,C 180,E1 -26683.925,E2 -26683.925} C_VEL
LIN {X 0,Y 106.293,Z 556.846,A -85,B 0,C 180,E1 -26685.719,E2 -26685.719} C_VEL
LIN {X 0,Y 106.037,Z 570.573,A -85,B 0,C 180,E1 -26688.488,E2 -26688.488} C_VEL
LIN {X 0,Y 105.493,Z 583.767,A -85,B 0,C 180,E1 -26691.958,E2 -26691.958} C_VEL
LIN {X 0,Y 104.797,Z 595.484,A -85,B 0,C 180,E1 -26695.83,E2 -26695.83} C_VEL
LIN {X 0,Y 104.188,Z 605.4,A -85,B 0,C 180,E1 -26699.832,E2 -26699.832} C_VEL
LIN {X 0,Y 103.723,Z 613.751,A -85,B 0,C 180,E1 -26703.869,E2 -26703.869} C_VEL
LIN {X 0,Y 103.304,Z 621.018,A -85,B 0,C 180,E1 -26708.027,E2 -26708.027} C_VEL
LIN {X 0,Y 101.924,Z 628.051,A -85,B 0,C 180,E1 -26712.96,E2 -26712.96} C_VEL
LIN {X 0,Y 101.246,Z 634.954,A -85,B 0,C 180,E1 -26718.996,E2 -26718.996} C_VEL
LIN {X 0,Y 101.383,Z 639.539,A -85,B 0,C 180,E1 -26724.032,E2 -26724.032} C_VEL
LIN {X 0,Y 102.348,Z 643.879,A -85,B 0,C 180,E1 -26730.001,E2 -26730.001} C_VEL
LIN {X 0,Y 101.542,Z 645.654,A -85,B 0,C 180,E1 -26733.969,E2 -26733.969} C_VEL
LIN {X 0,Y 100.479,Z 647.772,A -85,B 0,C 180,E1 -26742.113,E2 -26742.113} C_VEL
LIN {X 0,Y 101.584,Z 648.58,A -85,B 0,C 180,E1 -26750.239,E2 -26750.239} C_VEL
LIN {X 0,Y 104.934,Z 648.15,A -85,B 0,C 180,E1 -26757.959,E2 -26757.959} C_VEL
LIN {X 0,Y 110.473,Z 646.525,A -85,B 0,C 180,E1 -26764.929,E2 -26764.929} C_VEL
LIN {X 0,Y 117.689,Z 643.661,A -85,B 0,C 180,E1 -26771.063,E2 -26771.063} C_VEL
LIN {X 0,Y 125.841,Z 639.434,A -85,B 0,C 180,E1 -26776.555,E2 -26776.555} C_VEL
LIN {X 0,Y 133.423,Z 634.828,A -85,B 0,C 180,E1 -26780.796,E2 -26780.796} C_VEL
LIN {X 0,Y 141.389,Z 628.989,A -85,B 0,C 180,E1 -26785.102,E2 -26785.102} C_VEL
LIN {X 0,Y 146.992,Z 624.277,A -85,B 0,C 180,E1 -26788.27,E2 -26788.27} C_VEL
LIN {X 0,Y 147.761,Z 623.492,A -85,B 0,C 180,E1 -26788.887,E2 -26788.887} C_VEL
LIN {X 0,Y 148.636,Z 621.492,A -85,B 0,C 180,E1 -26791.782,E2 -26791.782} C_VEL
LIN {X 0,Y 149.214,Z 619.846,A -85,B 0,C 180,E1 -26794.919,E2 -26794.919} C_VEL
LIN {X 0,Y 149.932,Z 618.102,A -85,B 0,C 180,E1 -26799.636,E2 -26799.636} C_VEL
LIN {X 0,Y 150.03,Z 617.811,A -85,B 0,C 180,E1 -26800.859,E2 -26800.859} C_VEL
LIN {X 0,Y 149.823,Z 617.657,A -85,B 0,C 180,E1 -26803.654,E2 -26803.654} C_VEL
LIN {X 0,Y 148.413,Z 618.318,A -85,B 0,C 180,E1 -26806.305,E2 -26806.305} C_VEL
LIN {X 0,Y 145.557,Z 619.801,A -85,B 0,C 180,E1 -26808.91,E2 -26808.91} C_VEL
LIN {X 0,Y 137.009,Z 623.533,A -85,B 0,C 180,E1 -26812.605,E2 -26812.605} C_VEL
LIN {X 0,Y 126.562,Z 626.593,A -85,B 0,C 180,E1 -26818.29,E2 -26818.29} C_VEL
LIN {X 0,Y 119.397,Z 627.588,A -85,B 0,C 180,E1 -26823.375,E2 -26823.375} C_VEL
LIN {X 0,Y 113.701,Z 627.432,A -85,B 0,C 180,E1 -26828.51,E2 -26828.51} C_VEL
LIN {X 0,Y 108.015,Z 625.814,A -85,B 0,C 180,E1 -26835.524,E2 -26835.524} C_VEL
LIN {X 0,Y 105.106,Z 623.886,A -85,B 0,C 180,E1 -26840.588,E2 -26840.588} C_VEL
LIN {X 0,Y 102.639,Z 620.479,A -85,B 0,C 180,E1 -26847.106,E2 -26847.106} C_VEL
LIN {X 0,Y 101.719,Z 617.683,A -85,B 0,C 180,E1 -26851.369,E2 -26851.369} C_VEL
LIN {X 0,Y 100.727,Z 615.47,A -85,B 0,C 180,E1 -26854.389,E2 -26854.389} C_VEL
LIN {X 0,Y 97.809,Z 611.358,A -85,B 0,C 180,E1 -26859.299,E2 -26859.299} C_VEL
LIN {X 0,Y 95.434,Z 606.566,A -85,B 0,C 180,E1 -26864.302,E2 -26864.302} C_VEL
LIN {X 0,Y 95.337,Z 603.264,A -85,B 0,C 180,E1 -26867.311,E2 -26867.311} C_VEL
LIN {X 0,Y 97.54,Z 594.564,A -85,B 0,C 180,E1 -26873.872,E2 -26873.872} C_VEL
LIN {X 0,Y 100.195,Z 585.151,A -85,B 0,C 180,E1 -26879.454,E2 -26879.454} C_VEL
LIN {X 0,Y 103.009,Z 575.656,A -85,B 0,C 180,E1 -26883.906,E2 -26883.906} C_VEL
LIN {X 0,Y 104.157,Z 571.68,A -85,B 0,C 180,E1 -26885.485,E2 -26885.485} C_VEL
LIN {X 0,Y 102.58,Z 564.14,A -85,B 0,C 180,E1 -26888.918,E2 -26888.918} C_VEL
LIN {X 0,Y 99.96,Z 554.119,A -85,B 0,C 180,E1 -26893.201,E2 -26893.201} C_VEL
LIN {X 0,Y 97.003,Z 544.874,A -85,B 0,C 180,E1 -26896.903,E2 -26896.903} C_VEL
LIN {X 0,Y 94.139,Z 536.76,A -85,B 0,C 180,E1 -26900.058,E2 -26900.058} C_VEL
LIN {X 0,Y 94.775,Z 536.679,A -85,B 0,C 180,E1 -26909.999,E2 -26909.999} C_VEL
LIN {X 0,Y 94.167,Z 536.747,A -85,B 0,C 180,E1 -26918.584,E2 -26918.584} C_VEL
LIN {X 0,Y 94.014,Z 536.774,A -85,B 0,C 180,E1 -26923.63,E2 -26923.63} C_VEL
LIN {X 0,Y 93.695,Z 536.814,A -85,B 0,C 180,E1 -26932.027,E2 -26932.027} C_VEL
LIN {X 0,Y 93.621,Z 536.816,A -85,B 0,C 180,E1 -26936.769,E2 -26936.769} C_VEL
LIN {X 0,Y 93.586,Z 536.819,A -85,B 0,C 180,E1 -26944.301,E2 -26944.301} C_VEL
LIN {X 0,Y 93.529,Z 536.827,A -85,B 0,C 180,E1 -26952.553,E2 -26952.553} C_VEL
LIN {X 0,Y 93.535,Z 536.833,A -85,B 0,C 180,E1 -26958.709,E2 -26958.709} C_VEL
LIN {X 0,Y 93.594,Z 536.826,A -85,B 0,C 180,E1 -26965.689,E2 -26965.689} C_VEL
LIN {X 0,Y 93.67,Z 536.817,A -85,B 0,C 180,E1 -26974.203,E2 -26974.203} C_VEL
LIN {X 0,Y 93.693,Z 536.807,A -85,B 0,C 180,E1 -26977.971,E2 -26977.971} C_VEL
LIN {X 0,Y 94.022,Z 536.767,A -85,B 0,C 180,E1 -26986.344,E2 -26986.344} C_VEL
LIN {X 0,Y 94.174,Z 536.754,A -85,B 0,C 180,E1 -26991.415,E2 -26991.415} C_VEL
LIN {X 0,Y 94.77,Z 536.68,A -85,B 0,C 180,E1 -26999.999,E2 -26999.999} C_VEL
LIN {X 0,Y 94.161,Z 536.756,A -85,B 0,C 180,E1 -27008.584,E2 -27008.584} C_VEL
LIN {X 0,Y 94.001,Z 536.769,A -85,B 0,C 180,E1 -27013.605,E2 -27013.605} C_VEL
LIN {X 0,Y 93.69,Z 536.807,A -85,B 0,C 180,E1 -27022.027,E2 -27022.027} C_VEL
LIN {X 0,Y 93.86,Z 536.939,A -85,B 0,C 180,E1 -27029.739,E2 -27029.739} C_VEL
LIN {X 0,Y 94.652,Z 540.37,A -85,B 0,C 180,E1 -27035.239,E2 -27035.239} C_VEL
LIN {X 0,Y 95.507,Z 544.198,A -85,B 0,C 180,E1 -27040.773,E2 -27040.773} C_VEL
LIN {X 0,Y 98.013,Z 552.147,A -85,B 0,C 180,E1 -27042.792,E2 -27042.792} C_VEL
LIN {X 0,Y 99.732,Z 558.22,A -85,B 0,C 180,E1 -27044.377,E2 -27044.377} C_VEL
LIN {X 0,Y 99.32,Z 571.632,A -85,B 0,C 180,E1 -27047.373,E2 -27047.373} C_VEL
LIN {X 0,Y 98.599,Z 584.941,A -85,B 0,C 180,E1 -27051.249,E2 -27051.249} C_VEL
LIN {X 0,Y 97.737,Z 596.551,A -85,B 0,C 180,E1 -27055.51,E2 -27055.51} C_VEL
LIN {X 0,Y 97.008,Z 607.244,A -85,B 0,C 180,E1 -27060.385,E2 -27060.385} C_VEL
LIN {X 0,Y 96.509,Z 616.033,A -85,B 0,C 180,E1 -27065.246,E2 -27065.246} C_VEL
LIN {X 0,Y 96.115,Z 621.173,A -85,B 0,C 180,E1 -27068.556,E2 -27068.556} C_VEL
LIN {X 0,Y 94.5,Z 629.444,A -85,B 0,C 180,E1 -27075.196,E2 -27075.196} C_VEL
LIN {X 0,Y 94.277,Z 635.569,A -85,B 0,C 180,E1 -27081.426,E2 -27081.426} C_VEL
LIN {X 0,Y 94.981,Z 640.572,A -85,B 0,C 180,E1 -27087.88,E2 -27087.88} C_VEL
LIN {X 0,Y 95.372,Z 641.948,A -85,B 0,C 180,E1 -27090.001,E2 -27090.001} C_VEL
LIN {X 0,Y 94.634,Z 643.822,A -85,B 0,C 180,E1 -27094.26,E2 -27094.26} C_VEL
LIN {X 0,Y 93.614,Z 646.182,A -85,B 0,C 180,E1 -27103.017,E2 -27103.017} C_VEL
LIN {X 0,Y 94.969,Z 647.219,A -85,B 0,C 180,E1 -27111.717,E2 -27111.717} C_VEL
LIN {X 0,Y 98.698,Z 647.027,A -85,B 0,C 180,E1 -27119.898,E2 -27119.898} C_VEL
LIN {X 0,Y 104.731,Z 645.649,A -85,B 0,C 180,E1 -27127.154,E2 -27127.154} C_VEL
LIN {X 0,Y 112.379,Z 643.033,A -85,B 0,C 180,E1 -27133.467,E2 -27133.467} C_VEL
LIN {X 0,Y 121.014,Z 639.157,A -85,B 0,C 180,E1 -27139.025,E2 -27139.025} C_VEL
LIN {X 0,Y 128.279,Z 635.22,A -85,B 0,C 180,E1 -27142.94,E2 -27142.94} C_VEL
LIN {X 0,Y 137.31,Z 629.362,A -85,B 0,C 180,E1 -27147.622,E2 -27147.622} C_VEL
LIN {X 0,Y 139.631,Z 627.697,A -85,B 0,C 180,E1 -27148.834,E2 -27148.834} C_VEL
LIN {X 0,Y 141.836,Z 625.863,A -85,B 0,C 180,E1 -27150.298,E2 -27150.298} C_VEL
LIN {X 0,Y 142.713,Z 623.945,A -85,B 0,C 180,E1 -27153.692,E2 -27153.692} C_VEL
LIN {X 0,Y 143.534,Z 621.971,A -85,B 0,C 180,E1 -27158.485,E2 -27158.485} C_VEL
LIN {X 0,Y 143.754,Z 621.511,A -85,B 0,C 180,E1 -27159.988,E2 -27159.988} C_VEL
LIN {X 0,Y 143.631,Z 621.097,A -85,B 0,C 180,E1 -27162.928,E2 -27162.928} C_VEL
LIN {X 0,Y 142.059,Z 621.595,A -85,B 0,C 180,E1 -27165.679,E2 -27165.679} C_VEL
LIN {X 0,Y 137.638,Z 623.416,A -85,B 0,C 180,E1 -27168.215,E2 -27168.215} C_VEL
LIN {X 0,Y 131.637,Z 625.574,A -85,B 0,C 180,E1 -27170.784,E2 -27170.784} C_VEL
LIN {X 0,Y 125.989,Z 627.161,A -85,B 0,C 180,E1 -27173.595,E2 -27173.595} C_VEL
LIN {X 0,Y 119.615,Z 628.375,A -85,B 0,C 180,E1 -27177.252,E2 -27177.252} C_VEL
LIN {X 0,Y 110.941,Z 628.848,A -85,B 0,C 180,E1 -27183.633,E2 -27183.633} C_VEL
LIN {X 0,Y 106.439,Z 628.284,A -85,B 0,C 180,E1 -27187.929,E2 -27187.929} C_VEL
LIN {X 0,Y 101.451,Z 626.629,A -85,B 0,C 180,E1 -27194.103,E2 -27194.103} C_VEL
LIN {X 0,Y 97.582,Z 623.747,A -85,B 0,C 180,E1 -27201.108,E2 -27201.108} C_VEL
LIN {X 0,Y 94.942,Z 619.038,A -85,B 0,C 180,E1 -27209.387,E2 -27209.387} C_VEL
LIN {X 0,Y 94.181,Z 613.693,A -85,B 0,C 180,E1 -27216.655,E2 -27216.655} C_VEL
LIN {X 0,Y 94.595,Z 607.501,A -85,B 0,C 180,E1 -27223.414,E2 -27223.414} C_VEL
LIN {X 0,Y 95.337,Z 603.264,A -85,B 0,C 180,E1 -27227.311,E2 -27227.311} C_VEL
LIN {X 0,Y 95.4,Z 599.836,A -85,B 0,C 180,E1 -27230.207,E2 -27230.207} C_VEL
LIN {X 0,Y 94.1,Z 593.734,A -85,B 0,C 180,E1 -27234.885,E2 -27234.885} C_VEL
LIN {X 0,Y 93.29,Z 587.117,A -85,B 0,C 180,E1 -27239.388,E2 -27239.388} C_VEL
LIN {X 0,Y 94.094,Z 582.776,A -85,B 0,C 180,E1 -27241.84,E2 -27241.84} C_VEL
LIN {X 0,Y 97.294,Z 572.414,A -85,B 0,C 180,E1 -27246.59,E2 -27246.59} C_VEL
LIN {X 0,Y 95.182,Z 563.073,A -85,B 0,C 180,E1 -27251.153,E2 -27251.153} C_VEL
LIN {X 0,Y 92.467,Z 552.994,A -85,B 0,C 180,E1 -27255.698,E2 -27255.698} C_VEL
LIN {X 0,Y 88.864,Z 542.418,A -85,B 0,C 180,E1 -27260.324,E2 -27260.324} C_VEL
LIN {X 0,Y 87.127,Z 537.632,A -85,B 0,C 180,E1 -27262.467,E2 -27262.467} C_VEL
LIN {X 0,Y 87.704,Z 537.56,A -85,B 0,C 180,E1 -27269.999,E2 -27269.999} C_VEL
LIN {X 0,Y 87.077,Z 537.631,A -85,B 0,C 180,E1 -27279.289,E2 -27279.289} C_VEL
LIN {X 0,Y 86.934,Z 537.655,A -85,B 0,C 180,E1 -27284.035,E2 -27284.035} C_VEL
LIN {X 0,Y 86.646,Z 537.687,A -85,B 0,C 180,E1 -27288.932,E2 -27288.932} C_VEL
LIN {X 0,Y 86.585,Z 537.692,A -85,B 0,C 180,E1 -27296.762,E2 -27296.762} C_VEL
LIN {X 0,Y 86.504,Z 537.704,A -85,B 0,C 180,E1 -27305.662,E2 -27305.662} C_VEL
LIN {X 0,Y 86.453,Z 537.708,A -85,B 0,C 180,E1 -27312.974,E2 -27312.974} C_VEL
LIN {X 0,Y 86.457,Z 537.712,A -85,B 0,C 180,E1 -27319.433,E2 -27319.433} C_VEL
LIN {X 0,Y 86.537,Z 537.706,A -85,B 0,C 180,E1 -27325.353,E2 -27325.353} C_VEL
LIN {X 0,Y 86.586,Z 537.699,A -85,B 0,C 180,E1 -27333.232,E2 -27333.232} C_VEL
LIN {X 0,Y 86.646,Z 537.689,A -85,B 0,C 180,E1 -27341.066,E2 -27341.066} C_VEL
LIN {X 0,Y 86.932,Z 537.651,A -85,B 0,C 180,E1 -27345.962,E2 -27345.962} C_VEL
LIN {X 0,Y 87.084,Z 537.637,A -85,B 0,C 180,E1 -27350.71,E2 -27350.71} C_VEL
LIN {X 0,Y 87.7,Z 537.561,A -85,B 0,C 180,E1 -27359.999,E2 -27359.999} C_VEL
LIN {X 0,Y 87.073,Z 537.638,A -85,B 0,C 180,E1 -27369.289,E2 -27369.289} C_VEL
LIN {X 0,Y 86.895,Z 537.655,A -85,B 0,C 180,E1 -27374.041,E2 -27374.041} C_VEL
LIN {X 0,Y 86.63,Z 537.692,A -85,B 0,C 180,E1 -27378.934,E2 -27378.934} C_VEL
LIN {X 0,Y 86.671,Z 537.688,A -85,B 0,C 180,E1 -27386.878,E2 -27386.878} C_VEL
LIN {X 0,Y 86.785,Z 537.75,A -85,B 0,C 180,E1 -27389.402,E2 -27389.402} C_VEL
LIN {X 0,Y 87.814,Z 542.112,A -85,B 0,C 180,E1 -27396.839,E2 -27396.839} C_VEL
LIN {X 0,Y 87.924,Z 542.738,A -85,B 0,C 180,E1 -27397.859,E2 -27397.859} C_VEL
LIN {X 0,Y 89.231,Z 546.821,A -85,B 0,C 180,E1 -27399.056,E2 -27399.056} C_VEL
LIN {X 0,Y 92.584,Z 557.784,A -85,B 0,C 180,E1 -27402.352,E2 -27402.352} C_VEL
LIN {X 0,Y 93.167,Z 560.446,A -85,B 0,C 180,E1 -27403.126,E2 -27403.126} C_VEL
LIN {X 0,Y 92.426,Z 574.799,A -85,B 0,C 180,E1 -27406.816,E2 -27406.816} C_VEL
LIN {X 0,Y 91.573,Z 587.296,A -85,B 0,C 180,E1 -27411.019,E2 -27411.019} C_VEL
LIN {X 0,Y 90.606,Z 598.694,A -85,B 0,C 180,E1 -27415.782,E2 -27415.782} C_VEL
LIN {X 0,Y 89.827,Z 608.897,A -85,B 0,C 180,E1 -27421.054,E2 -27421.054} C_VEL
LIN {X 0,Y 89.29,Z 617.971,A -85,B 0,C 180,E1 -27426.825,E2 -27426.825} C_VEL
LIN {X 0,Y 88.587,Z 622.545,A -85,B 0,C 180,E1 -27430.296,E2 -27430.296} C_VEL
LIN {X 0,Y 87.388,Z 630.035,A -85,B 0,C 180,E1 -27437.223,E2 -27437.223} C_VEL
LIN {X 0,Y 87.42,Z 635.102,A -85,B 0,C 180,E1 -27443.074,E2 -27443.074} C_VEL
LIN {X 0,Y 88.395,Z 639.943,A -85,B 0,C 180,E1 -27450.001,E2 -27450.001} C_VEL
LIN {X 0,Y 87.701,Z 641.981,A -85,B 0,C 180,E1 -27454.597,E2 -27454.597} C_VEL
LIN {X 0,Y 86.778,Z 644.513,A -85,B 0,C 180,E1 -27464.062,E2 -27464.062} C_VEL
LIN {X 0,Y 88.429,Z 645.763,A -85,B 0,C 180,E1 -27473.415,E2 -27473.415} C_VEL
LIN {X 0,Y 92.612,Z 645.816,A -85,B 0,C 180,E1 -27482.088,E2 -27482.088} C_VEL
LIN {X 0,Y 99.149,Z 644.722,A -85,B 0,C 180,E1 -27489.64,E2 -27489.64} C_VEL
LIN {X 0,Y 107.294,Z 642.412,A -85,B 0,C 180,E1 -27496.099,E2 -27496.099} C_VEL
LIN {X 0,Y 116.418,Z 638.831,A -85,B 0,C 180,E1 -27501.703,E2 -27501.703} C_VEL
LIN {X 0,Y 123.345,Z 635.527,A -85,B 0,C 180,E1 -27505.266,E2 -27505.266} C_VEL
LIN {X 0,Y 131.054,Z 631.189,A -85,B 0,C 180,E1 -27509.097,E2 -27509.097} C_VEL
LIN {X 0,Y 133.488,Z 629.66,A -85,B 0,C 180,E1 -27510.31,E2 -27510.31} C_VEL
LIN {X 0,Y 135.683,Z 628.138,A -85,B 0,C 180,E1 -27511.711,E2 -27511.711} C_VEL
LIN {X 0,Y 136.918,Z 625.512,A -85,B 0,C 180,E1 -27517.51,E2 -27517.51} C_VEL
LIN {X 0,Y 137.222,Z 624.989,A -85,B 0,C 180,E1 -27518.992,E2 -27518.992} C_VEL
LIN {X 0,Y 137.258,Z 624.306,A -85,B 0,C 180,E1 -27522.109,E2 -27522.109} C_VEL
LIN {X 0,Y 135.101,Z 624.817,A -85,B 0,C 180,E1 -27524.925,E2 -27524.925} C_VEL
LIN {X 0,Y 129.591,Z 626.649,A -85,B 0,C 180,E1 -27527.472,E2 -27527.472} C_VEL
LIN {X 0,Y 120.813,Z 628.845,A -85,B 0,C 180,E1 -27531.475,E2 -27531.475} C_VEL
LIN {X 0,Y 112.197,Z 629.992,A -85,B 0,C 180,E1 -27536.41,E2 -27536.41} C_VEL
LIN {X 0,Y 105.449,Z 630,A -85,B 0,C 180,E1 -27541.299,E2 -27541.299} C_VEL
LIN {X 0,Y 98.304,Z 628.721,A -85,B 0,C 180,E1 -27548.222,E2 -27548.222} C_VEL
LIN {X 0,Y 94.091,Z 626.882,A -85,B 0,C 180,E1 -27553.825,E2 -27553.825} C_VEL
LIN {X 0,Y 90.316,Z 623.732,A -85,B 0,C 180,E1 -27560.965,E2 -27560.965} C_VEL
LIN {X 0,Y 87.969,Z 619.409,A -85,B 0,C 180,E1 -27568.645,E2 -27568.645} C_VEL
LIN {X 0,Y 87.117,Z 614.085,A -85,B 0,C 180,E1 -27576.221,E2 -27576.221} C_VEL
LIN {X 0,Y 87.509,Z 607.533,A -85,B 0,C 180,E1 -27583.713,E2 -27583.713} C_VEL
LIN {X 0,Y 89.191,Z 599.582,A -85,B 0,C 180,E1 -27590.921,E2 -27590.921} C_VEL
LIN {X 0,Y 91.786,Z 590.243,A -85,B 0,C 180,E1 -27597.588,E2 -27597.588} C_VEL
LIN {X 0,Y 94.094,Z 582.776,A -85,B 0,C 180,E1 -27601.84,E2 -27601.84} C_VEL
LIN {X 0,Y 94.37,Z 579.89,A -85,B 0,C 180,E1 -27603.416,E2 -27603.416} C_VEL
LIN {X 0,Y 93.59,Z 577.091,A -85,B 0,C 180,E1 -27605.065,E2 -27605.065} C_VEL
LIN {X 0,Y 89.406,Z 568.723,A -85,B 0,C 180,E1 -27610.163,E2 -27610.163} C_VEL
LIN {X 0,Y 89.113,Z 567.676,A -85,B 0,C 180,E1 -27610.716,E2 -27610.716} C_VEL
LIN {X 0,Y 86.596,Z 557.407,A -85,B 0,C 180,E1 -27615.907,E2 -27615.907} C_VEL
LIN {X 0,Y 83.444,Z 547.166,A -85,B 0,C 180,E1 -27620.913,E2 -27620.913} C_VEL
LIN {X 0,Y 80.196,Z 538.832,A -85,B 0,C 180,E1 -27624.972,E2 -27624.972} C_VEL
LIN {X 0,Y 80.165,Z 538.499,A -85,B 0,C 180,E1 -27625.285,E2 -27625.285} C_VEL
LIN {X 0,Y 80.633,Z 538.441,A -85,B 0,C 180,E1 -27629.999,E2 -27629.999} C_VEL
LIN {X 0,Y 79.962,Z 538.519,A -85,B 0,C 180,E1 -27640.124,E2 -27640.124} C_VEL
LIN {X 0,Y 79.746,Z 538.547,A -85,B 0,C 180,E1 -27645.33,E2 -27645.33} C_VEL
LIN {X 0,Y 79.514,Z 538.58,A -85,B 0,C 180,E1 -27650.704,E2 -27650.704} C_VEL
LIN {X 0,Y 79.482,Z 538.581,A -85,B 0,C 180,E1 -27657.84,E2 -27657.84} C_VEL
LIN {X 0,Y 79.385,Z 538.595,A -85,B 0,C 180,E1 -27667.174,E2 -27667.174} C_VEL
LIN {X 0,Y 79.383,Z 538.593,A -85,B 0,C 180,E1 -27675.093,E2 -27675.093} C_VEL
LIN {X 0,Y 79.389,Z 538.59,A -85,B 0,C 180,E1 -27682.819,E2 -27682.819} C_VEL
LIN {X 0,Y 79.382,Z 538.594,A -85,B 0,C 180,E1 -27687.911,E2 -27687.911} C_VEL
LIN {X 0,Y 79.527,Z 538.579,A -85,B 0,C 180,E1 -27693.775,E2 -27693.775} C_VEL
LIN {X 0,Y 79.514,Z 538.573,A -85,B 0,C 180,E1 -27699.294,E2 -27699.294} C_VEL
LIN {X 0,Y 79.825,Z 538.537,A -85,B 0,C 180,E1 -27705.571,E2 -27705.571} C_VEL
LIN {X 0,Y 79.967,Z 538.523,A -85,B 0,C 180,E1 -27709.875,E2 -27709.875} C_VEL
LIN {X 0,Y 80.629,Z 538.441,A -85,B 0,C 180,E1 -27719.999,E2 -27719.999} C_VEL
LIN {X 0,Y 79.953,Z 538.525,A -85,B 0,C 180,E1 -27730.124,E2 -27730.124} C_VEL
LIN {X 0,Y 79.727,Z 538.551,A -85,B 0,C 180,E1 -27735.333,E2 -27735.333} C_VEL
LIN {X 0,Y 79.51,Z 538.573,A -85,B 0,C 180,E1 -27740.704,E2 -27740.704} C_VEL
LIN {X 0,Y 79.731,Z 538.615,A -85,B 0,C 180,E1 -27749.164,E2 -27749.164} C_VEL
LIN {X 0,Y 80.442,Z 541.506,A -85,B 0,C 180,E1 -27754.602,E2 -27754.602} C_VEL
LIN {X 0,Y 81.645,Z 545.393,A -85,B 0,C 180,E1 -27755.902,E2 -27755.902} C_VEL
LIN {X 0,Y 84.838,Z 554.895,A -85,B 0,C 180,E1 -27759.191,E2 -27759.191} C_VEL
LIN {X 0,Y 86.645,Z 561.973,A -85,B 0,C 180,E1 -27761.562,E2 -27761.562} C_VEL
LIN {X 0,Y 85.727,Z 575.169,A -85,B 0,C 180,E1 -27765.359,E2 -27765.359} C_VEL
LIN {X 0,Y 84.667,Z 587.595,A -85,B 0,C 180,E1 -27769.962,E2 -27769.962} C_VEL
LIN {X 0,Y 83.594,Z 598.637,A -85,B 0,C 180,E1 -27775.052,E2 -27775.052} C_VEL
LIN {X 0,Y 82.749,Z 608.622,A -85,B 0,C 180,E1 -27780.768,E2 -27780.768} C_VEL
LIN {X 0,Y 82.296,Z 616.319,A -85,B 0,C 180,E1 -27786.069,E2 -27786.069} C_VEL
LIN {X 0,Y 81.696,Z 621.009,A -85,B 0,C 180,E1 -27789.873,E2 -27789.873} C_VEL
LIN {X 0,Y 80.438,Z 628.56,A -85,B 0,C 180,E1 -27797.384,E2 -27797.384} C_VEL
LIN {X 0,Y 80.637,Z 634.621,A -85,B 0,C 180,E1 -27805.001,E2 -27805.001} C_VEL
LIN {X 0,Y 81.415,Z 637.861,A -85,B 0,C 180,E1 -27810.001,E2 -27810.001} C_VEL
LIN {X 0,Y 81.237,Z 639.074,A -85,B 0,C 180,E1 -27812.48,E2 -27812.48} C_VEL
LIN {X 0,Y 80.054,Z 641.566,A -85,B 0,C 180,E1 -27820.113,E2 -27820.113} C_VEL
LIN {X 0,Y 80.64,Z 643.701,A -85,B 0,C 180,E1 -27830.403,E2 -27830.403} C_VEL
LIN {X 0,Y 84.02,Z 644.574,A -85,B 0,C 180,E1 -27840.125,E2 -27840.125} C_VEL
LIN {X 0,Y 89.966,Z 644.296,A -85,B 0,C 180,E1 -27848.679,E2 -27848.679} C_VEL
LIN {X 0,Y 97.992,Z 642.867,A -85,B 0,C 180,E1 -27855.825,E2 -27855.825} C_VEL
LIN {X 0,Y 107.153,Z 640.194,A -85,B 0,C 180,E1 -27861.913,E2 -27861.913} C_VEL
LIN {X 0,Y 117.188,Z 636.35,A -85,B 0,C 180,E1 -27867.1,E2 -27867.1} C_VEL
LIN {X 0,Y 124.856,Z 632.694,A -85,B 0,C 180,E1 -27870.75,E2 -27870.75} C_VEL
LIN {X 0,Y 128.921,Z 630.494,A -85,B 0,C 180,E1 -27872.743,E2 -27872.743} C_VEL
LIN {X 0,Y 129.594,Z 629.684,A -85,B 0,C 180,E1 -27874.289,E2 -27874.289} C_VEL
LIN {X 0,Y 130.4,Z 628.239,A -85,B 0,C 180,E1 -27877.836,E2 -27877.836} C_VEL
LIN {X 0,Y 130.687,Z 627.285,A -85,B 0,C 180,E1 -27881.177,E2 -27881.177} C_VEL
LIN {X 0,Y 127.636,Z 627.873,A -85,B 0,C 180,E1 -27884.02,E2 -27884.02} C_VEL
LIN {X 0,Y 121.476,Z 629.414,A -85,B 0,C 180,E1 -27886.62,E2 -27886.62} C_VEL
LIN {X 0,Y 114.195,Z 630.734,A -85,B 0,C 180,E1 -27889.968,E2 -27889.968} C_VEL
LIN {X 0,Y 105.873,Z 631.356,A -85,B 0,C 180,E1 -27894.705,E2 -27894.705} C_VEL
LIN {X 0,Y 98.394,Z 630.955,A -85,B 0,C 180,E1 -27900.125,E2 -27900.125} C_VEL
LIN {X 0,Y 91.937,Z 629.488,A -85,B 0,C 180,E1 -27906.392,E2 -27906.392} C_VEL
LIN {X 0,Y 86.307,Z 626.686,A -85,B 0,C 180,E1 -27914.141,E2 -27914.141} C_VEL
LIN {X 0,Y 82.224,Z 622.359,A -85,B 0,C 180,E1 -27923.158,E2 -27923.158} C_VEL
LIN {X 0,Y 80.357,Z 617.235,A -85,B 0,C 180,E1 -27931.654,E2 -27931.654} C_VEL
LIN {X 0,Y 80.112,Z 610.056,A -85,B 0,C 180,E1 -27941.146,E2 -27941.146} C_VEL
LIN {X 0,Y 81.491,Z 602.183,A -85,B 0,C 180,E1 -27949.358,E2 -27949.358} C_VEL
LIN {X 0,Y 84.063,Z 593.024,A -85,B 0,C 180,E1 -27956.727,E2 -27956.727} C_VEL
LIN {X 0,Y 87.459,Z 582.295,A -85,B 0,C 180,E1 -27963.381,E2 -27963.381} C_VEL
LIN {X 0,Y 90.342,Z 573.28,A -85,B 0,C 180,E1 -27967.713,E2 -27967.713} C_VEL
LIN {X 0,Y 89.113,Z 567.676,A -85,B 0,C 180,E1 -27970.716,E2 -27970.716} C_VEL
LIN {X 0,Y 87.501,Z 563.37,A -85,B 0,C 180,E1 -27973.12,E2 -27973.12} C_VEL
LIN {X 0,Y 84.994,Z 559.478,A -85,B 0,C 180,E1 -27975.602,E2 -27975.602} C_VEL
LIN {X 0,Y 77.425,Z 549.377,A -85,B 0,C 180,E1 -27982.619,E2 -27982.619} C_VEL
LIN {X 0,Y 75.969,Z 546.474,A -85,B 0,C 180,E1 -27984.387,E2 -27984.387} C_VEL
LIN {X 0,Y 73.468,Z 540.159,A -85,B 0,C 180,E1 -27987.943,E2 -27987.943} C_VEL
LIN {X 0,Y 73.364,Z 539.345,A -85,B 0,C 180,E1 -27988.455,E2 -27988.455} C_VEL
LIN {X 0,Y 73.561,Z 539.322,A -85,B 0,C 180,E1 -27989.999,E2 -27989.999} C_VEL
LIN {X 0,Y 72.856,Z 539.407,A -85,B 0,C 180,E1 -28001.123,E2 -28001.123} C_VEL
LIN {X 0,Y 72.576,Z 539.436,A -85,B 0,C 180,E1 -28006.888,E2 -28006.888} C_VEL
LIN {X 0,Y 72.395,Z 539.466,A -85,B 0,C 180,E1 -28012.849,E2 -28012.849} C_VEL
LIN {X 0,Y 72.359,Z 539.471,A -85,B 0,C 180,E1 -28019.053,E2 -28019.053} C_VEL
LIN {X 0,Y 72.293,Z 539.473,A -85,B 0,C 180,E1 -28025.682,E2 -28025.682} C_VEL
LIN {X 0,Y 72.244,Z 539.477,A -85,B 0,C 180,E1 -28032.919,E2 -28032.919} C_VEL
LIN {X 0,Y 72.295,Z 539.471,A -85,B 0,C 180,E1 -28041.05,E2 -28041.05} C_VEL
LIN {X 0,Y 72.297,Z 539.478,A -85,B 0,C 180,E1 -28044.318,E2 -28044.318} C_VEL
LIN {X 0,Y 72.376,Z 539.461,A -85,B 0,C 180,E1 -28050.951,E2 -28050.951} C_VEL
LIN {X 0,Y 72.395,Z 539.462,A -85,B 0,C 180,E1 -28057.149,E2 -28057.149} C_VEL
LIN {X 0,Y 72.722,Z 539.423,A -85,B 0,C 180,E1 -28065.108,E2 -28065.108} C_VEL
LIN {X 0,Y 72.858,Z 539.404,A -85,B 0,C 180,E1 -28068.875,E2 -28068.875} C_VEL
LIN {X 0,Y 73.556,Z 539.322,A -85,B 0,C 180,E1 -28079.999,E2 -28079.999} C_VEL
LIN {X 0,Y 72.844,Z 539.407,A -85,B 0,C 180,E1 -28091.124,E2 -28091.124} C_VEL
LIN {X 0,Y 72.565,Z 539.446,A -85,B 0,C 180,E1 -28096.89,E2 -28096.89} C_VEL
LIN {X 0,Y 72.692,Z 539.439,A -85,B 0,C 180,E1 -28108.907,E2 -28108.907} C_VEL
LIN {X 0,Y 72.862,Z 540.208,A -85,B 0,C 180,E1 -28110.537,E2 -28110.537} C_VEL
LIN {X 0,Y 74.263,Z 544.348,A -85,B 0,C 180,E1 -28112.188,E2 -28112.188} C_VEL
LIN {X 0,Y 75.121,Z 546.51,A -85,B 0,C 180,E1 -28113.151,E2 -28113.151} C_VEL
LIN {X 0,Y 78.403,Z 556.65,A -85,B 0,C 180,E1 -28117.232,E2 -28117.232} C_VEL
LIN {X 0,Y 80.061,Z 563.747,A -85,B 0,C 180,E1 -28119.95,E2 -28119.95} C_VEL
LIN {X 0,Y 78.813,Z 577.627,A -85,B 0,C 180,E1 -28124.49,E2 -28124.49} C_VEL
LIN {X 0,Y 77.544,Z 589.996,A -85,B 0,C 180,E1 -28129.778,E2 -28129.778} C_VEL
LIN {X 0,Y 76.325,Z 601.496,A -85,B 0,C 180,E1 -28135.966,E2 -28135.966} C_VEL
LIN {X 0,Y 75.528,Z 610.91,A -85,B 0,C 180,E1 -28142.274,E2 -28142.274} C_VEL
LIN {X 0,Y 75.015,Z 617.966,A -85,B 0,C 180,E1 -28147.992,E2 -28147.992} C_VEL
LIN {X 0,Y 73.599,Z 625.878,A -85,B 0,C 180,E1 -28156.189,E2 -28156.189} C_VEL
LIN {X 0,Y 73.673,Z 632.21,A -85,B 0,C 180,E1 -28164.527,E2 -28164.527} C_VEL
LIN {X 0,Y 74.44,Z 635.666,A -85,B 0,C 180,E1 -28170.001,E2 -28170.001} C_VEL
LIN {X 0,Y 74.438,Z 636.97,A -85,B 0,C 180,E1 -28172.706,E2 -28172.706} C_VEL
LIN {X 0,Y 73.233,Z 639.671,A -85,B 0,C 180,E1 -28181.067,E2 -28181.067} C_VEL
LIN {X 0,Y 74.113,Z 641.988,A -85,B 0,C 180,E1 -28192.292,E2 -28192.292} C_VEL
LIN {X 0,Y 78.015,Z 643.115,A -85,B 0,C 180,E1 -28202.719,E2 -28202.719} C_VEL
LIN {X 0,Y 84.568,Z 643.104,A -85,B 0,C 180,E1 -28211.671,E2 -28211.671} C_VEL
LIN {X 0,Y 93.158,Z 641.961,A -85,B 0,C 180,E1 -28218.976,E2 -28218.976} C_VEL
LIN {X 0,Y 102.888,Z 639.61,A -85,B 0,C 180,E1 -28225.055,E2 -28225.055} C_VEL
LIN {X 0,Y 114.009,Z 635.839,A -85,B 0,C 180,E1 -28230.453,E2 -28230.453} C_VEL
LIN {X 0,Y 121.412,Z 632.669,A -85,B 0,C 180,E1 -28233.797,E2 -28233.797} C_VEL
LIN {X 0,Y 123.182,Z 631.416,A -85,B 0,C 180,E1 -28235.906,E2 -28235.906} C_VEL
LIN {X 0,Y 123.847,Z 630.027,A -85,B 0,C 180,E1 -28240.094,E2 -28240.094} C_VEL
LIN {X 0,Y 122.572,Z 630.059,A -85,B 0,C 180,E1 -28241.702,E2 -28241.702} C_VEL
LIN {X 0,Y 119.928,Z 630.588,A -85,B 0,C 180,E1 -28242.963,E2 -28242.963} C_VEL
LIN {X 0,Y 113.318,Z 631.759,A -85,B 0,C 180,E1 -28245.637,E2 -28245.637} C_VEL
LIN {X 0,Y 106.926,Z 632.449,A -85,B 0,C 180,E1 -28248.629,E2 -28248.629} C_VEL
LIN {X 0,Y 99.11,Z 632.57,A -85,B 0,C 180,E1 -28253.105,E2 -28253.105} C_VEL
LIN {X 0,Y 89.982,Z 631.402,A -85,B 0,C 180,E1 -28260.001,E2 -28260.001} C_VEL
LIN {X 0,Y 84.713,Z 629.821,A -85,B 0,C 180,E1 -28265.4,E2 -28265.4} C_VEL
LIN {X 0,Y 79.339,Z 626.874,A -85,B 0,C 180,E1 -28272.989,E2 -28272.989} C_VEL
LIN {X 0,Y 75.35,Z 622.598,A -85,B 0,C 180,E1 -28281.908,E2 -28281.908} C_VEL
LIN {X 0,Y 73.382,Z 617.667,A -85,B 0,C 180,E1 -28290.462,E2 -28290.462} C_VEL
LIN {X 0,Y 72.986,Z 610.422,A -85,B 0,C 180,E1 -28300.73,E2 -28300.73} C_VEL
LIN {X 0,Y 74.261,Z 602.903,A -85,B 0,C 180,E1 -28309.213,E2 -28309.213} C_VEL
LIN {X 0,Y 76.638,Z 594.588,A -85,B 0,C 180,E1 -28316.617,E2 -28316.617} C_VEL
LIN {X 0,Y 79.722,Z 585.103,A -85,B 0,C 180,E1 -28323.202,E2 -28323.202} C_VEL
LIN {X 0,Y 83.087,Z 575.18,A -85,B 0,C 180,E1 -28328.509,E2 -28328.509} C_VEL
LIN {X 0,Y 83.242,Z 573.473,A -85,B 0,C 180,E1 -28329.408,E2 -28329.408} C_VEL
LIN {X 0,Y 81.129,Z 563.883,A -85,B 0,C 180,E1 -28334.936,E2 -28334.936} C_VEL
LIN {X 0,Y 78.823,Z 555.036,A -85,B 0,C 180,E1 -28339.727,E2 -28339.727} C_VEL
LIN {X 0,Y 75.969,Z 546.474,A -85,B 0,C 180,E1 -28344.387,E2 -28344.387} C_VEL
LIN {X 0,Y 74.164,Z 543.879,A -85,B 0,C 180,E1 -28346.305,E2 -28346.305} C_VEL
LIN {X 0,Y 71.763,Z 542.134,A -85,B 0,C 180,E1 -28348.524,E2 -28348.524} C_VEL
LIN {X 0,Y 68.515,Z 540.83,A -85,B 0,C 180,E1 -28352.032,E2 -28352.032} C_VEL
LIN {X 0,Y 66.178,Z 540.328,A -85,B 0,C 180,E1 -28356.295,E2 -28356.295} C_VEL
LIN {X 0,Y 65.752,Z 540.282,A -85,B 0,C 180,E1 -28358.664,E2 -28358.664} C_VEL
LIN {X 0,Y 65.62,Z 540.306,A -85,B 0,C 180,E1 -28365.432,E2 -28365.432} C_VEL
LIN {X 0,Y 65.231,Z 540.35,A -85,B 0,C 180,E1 -28375.528,E2 -28375.528} C_VEL
LIN {X 0,Y 65.17,Z 540.362,A -85,B 0,C 180,E1 -28382.628,E2 -28382.628} C_VEL
LIN {X 0,Y 65.18,Z 540.361,A -85,B 0,C 180,E1 -28390.991,E2 -28390.991} C_VEL
LIN {X 0,Y 65.201,Z 540.358,A -85,B 0,C 180,E1 -28399.702,E2 -28399.702} C_VEL
LIN {X 0,Y 65.255,Z 540.348,A -85,B 0,C 180,E1 -28409.496,E2 -28409.496} C_VEL
LIN {X 0,Y 65.24,Z 540.359,A -85,B 0,C 180,E1 -28414.473,E2 -28414.473} C_VEL
LIN {X 0,Y 65.626,Z 540.308,A -85,B 0,C 180,E1 -28424.541,E2 -28424.541} C_VEL
LIN {X 0,Y 65.755,Z 540.285,A -85,B 0,C 180,E1 -28427.655,E2 -28427.655} C_VEL
LIN {X 0,Y 66.481,Z 540.204,A -85,B 0,C 180,E1 -28439.998,E2 -28439.998} C_VEL
LIN {X 0,Y 65.742,Z 540.287,A -85,B 0,C 180,E1 -28452.344,E2 -28452.344} C_VEL
LIN {X 0,Y 65.383,Z 540.339,A -85,B 0,C 180,E1 -28458.811,E2 -28458.811} C_VEL
LIN {X 0,Y 65.489,Z 540.328,A -85,B 0,C 180,E1 -28465.845,E2 -28465.845} C_VEL
LIN {X 0,Y 66.625,Z 543.268,A -85,B 0,C 180,E1 -28467.483,E2 -28467.483} C_VEL
LIN {X 0,Y 67.658,Z 544.944,A -85,B 0,C 180,E1 -28468.615,E2 -28468.615} C_VEL
LIN {X 0,Y 69.976,Z 551.53,A -85,B 0,C 180,E1 -28471.821,E2 -28471.821} C_VEL
LIN {X 0,Y 72.392,Z 559.762,A -85,B 0,C 180,E1 -28475.625,E2 -28475.625} C_VEL
LIN {X 0,Y 73.563,Z 564.896,A -85,B 0,C 180,E1 -28477.923,E2 -28477.923} C_VEL
LIN {X 0,Y 72.131,Z 577.915,A -85,B 0,C 180,E1 -28482.704,E2 -28482.704} C_VEL
LIN {X 0,Y 70.591,Z 590.522,A -85,B 0,C 180,E1 -28488.733,E2 -28488.733} C_VEL
LIN {X 0,Y 69.333,Z 600.98,A -85,B 0,C 180,E1 -28495.027,E2 -28495.027} C_VEL
LIN {X 0,Y 68.408,Z 610.851,A -85,B 0,C 180,E1 -28502.464,E2 -28502.464} C_VEL
LIN {X 0,Y 68.061,Z 616.179,A -85,B 0,C 180,E1 -28507.232,E2 -28507.232} C_VEL
LIN {X 0,Y 66.81,Z 623.043,A -85,B 0,C 180,E1 -28514.754,E2 -28514.754} C_VEL
LIN {X 0,Y 66.747,Z 629.764,A -85,B 0,C 180,E1 -28523.957,E2 -28523.957} C_VEL
LIN {X 0,Y 67.475,Z 633.374,A -85,B 0,C 180,E1 -28530.001,E2 -28530.001} C_VEL
LIN {X 0,Y 67.644,Z 634.857,A -85,B 0,C 180,E1 -28532.979,E2 -28532.979} C_VEL
LIN {X 0,Y 66.458,Z 637.671,A -85,B 0,C 180,E1 -28542.211,E2 -28542.211} C_VEL
LIN {X 0,Y 67.698,Z 640.25,A -85,B 0,C 180,E1 -28554.536,E2 -28554.536} C_VEL
LIN {X 0,Y 72.192,Z 641.618,A -85,B 0,C 180,E1 -28565.741,E2 -28565.741} C_VEL
LIN {X 0,Y 79.433,Z 641.862,A -85,B 0,C 180,E1 -28575.059,E2 -28575.059} C_VEL
LIN {X 0,Y 88.64,Z 640.98,A -85,B 0,C 180,E1 -28582.456,E2 -28582.456} C_VEL
LIN {X 0,Y 98.959,Z 638.914,A -85,B 0,C 180,E1 -28588.457,E2 -28588.457} C_VEL
LIN {X 0,Y 109.97,Z 635.707,A -85,B 0,C 180,E1 -28593.474,E2 -28593.474} C_VEL
LIN {X 0,Y 115.536,Z 633.678,A -85,B 0,C 180,E1 -28595.847,E2 -28595.847} C_VEL
LIN {X 0,Y 116.779,Z 632.49,A -85,B 0,C 180,E1 -28598.833,E2 -28598.833} C_VEL
LIN {X 0,Y 115.416,Z 632.461,A -85,B 0,C 180,E1 -28600.434,E2 -28600.434} C_VEL
LIN {X 0,Y 105.143,Z 633.689,A -85,B 0,C 180,E1 -28604.493,E2 -28604.493} C_VEL
LIN {X 0,Y 98.626,Z 633.855,A -85,B 0,C 180,E1 -28607.657,E2 -28607.657} C_VEL
LIN {X 0,Y 92.44,Z 633.566,A -85,B 0,C 180,E1 -28611.255,E2 -28611.255} C_VEL
LIN {X 0,Y 84.442,Z 632.271,A -85,B 0,C 180,E1 -28617.142,E2 -28617.142} C_VEL
LIN {X 0,Y 76.657,Z 629.541,A -85,B 0,C 180,E1 -28625.262,E2 -28625.262} C_VEL
LIN {X 0,Y 70.766,Z 625.469,A -85,B 0,C 180,E1 -28634.794,E2 -28634.794} C_VEL
LIN {X 0,Y 67.297,Z 620.49,A -85,B 0,C 180,E1 -28644.693,E2 -28644.693} C_VEL
LIN {X 0,Y 65.839,Z 613.734,A -85,B 0,C 180,E1 -28655.954,E2 -28655.954} C_VEL
LIN {X 0,Y 66.453,Z 606.224,A -85,B 0,C 180,E1 -28665.979,E2 -28665.979} C_VEL
LIN {X 0,Y 68.998,Z 596.729,A -85,B 0,C 180,E1 -28675.856,E2 -28675.856} C_VEL
LIN {X 0,Y 72.43,Z 586.457,A -85,B 0,C 180,E1 -28683.841,E2 -28683.841} C_VEL
LIN {X 0,Y 76.339,Z 575.652,A -85,B 0,C 180,E1 -28690.133,E2 -28690.133} C_VEL
LIN {X 0,Y 75.187,Z 568.843,A -85,B 0,C 180,E1 -28694.41,E2 -28694.41} C_VEL
LIN {X 0,Y 72.948,Z 559.221,A -85,B 0,C 180,E1 -28700.293,E2 -28700.293} C_VEL
LIN {X 0,Y 70.225,Z 550.198,A -85,B 0,C 180,E1 -28705.832,E2 -28705.832} C_VEL
LIN {X 0,Y 67.859,Z 543.681,A -85,B 0,C 180,E1 -28709.999,E2 -28709.999} C_VEL
LIN {X 0,Y 66.654,Z 541.791,A -85,B 0,C 180,E1 -28711.51,E2 -28711.51} C_VEL
LIN {X 0,Y 66.172,Z 540.24,A -85,B 0,C 180,E1 -28712.662,E2 -28712.662} C_VEL
LIN {X 0,Y 65.752,Z 540.282,A -85,B 0,C 180,E1 -28718.664,E2 -28718.664} C_VEL
LIN {X 0,Y 65.332,Z 540.347,A -85,B 0,C 180,E1 -28722.08,E2 -28722.08} C_VEL
LIN {X 0,Y 63.898,Z 540.528,A -85,B 0,C 180,E1 -28727.178,E2 -28727.178} C_VEL
LIN {X 0,Y 61.976,Z 540.784,A -85,B 0,C 180,E1 -28732.324,E2 -28732.324} C_VEL
LIN {X 0,Y 58.003,Z 541.255,A -85,B 0,C 180,E1 -28747.623,E2 -28747.623} C_VEL
LIN {X 0,Y 58.011,Z 541.259,A -85,B 0,C 180,E1 -28756.626,E2 -28756.626} C_VEL
LIN {X 0,Y 58.031,Z 541.248,A -85,B 0,C 180,E1 -28762.73,E2 -28762.73} C_VEL
LIN {X 0,Y 58.159,Z 541.237,A -85,B 0,C 180,E1 -28767.766,E2 -28767.766} C_VEL
LIN {X 0,Y 58.151,Z 541.233,A -85,B 0,C 180,E1 -28771.088,E2 -28771.088} C_VEL
LIN {X 0,Y 58.517,Z 541.195,A -85,B 0,C 180,E1 -28783.905,E2 -28783.905} C_VEL
LIN {X 0,Y 58.798,Z 541.159,A -85,B 0,C 180,E1 -28793.133,E2 -28793.133} C_VEL
LIN {X 0,Y 59.371,Z 541.09,A -85,B 0,C 180,E1 -28799.998,E2 -28799.998} C_VEL
LIN {X 0,Y 58.788,Z 541.159,A -85,B 0,C 180,E1 -28806.864,E2 -28806.864} C_VEL
LIN {X 0,Y 58.503,Z 541.197,A -85,B 0,C 180,E1 -28816.047,E2 -28816.047} C_VEL
LIN {X 0,Y 58.291,Z 541.217,A -85,B 0,C 180,E1 -28820.164,E2 -28820.164} C_VEL
LIN {X 0,Y 59.331,Z 544.166,A -85,B 0,C 180,E1 -28822.181,E2 -28822.181} C_VEL
LIN {X 0,Y 60.949,Z 546.208,A -85,B 0,C 180,E1 -28824.253,E2 -28824.253} C_VEL
LIN {X 0,Y 62.579,Z 549.687,A -85,B 0,C 180,E1 -28826.692,E2 -28826.692} C_VEL
LIN {X 0,Y 64.769,Z 556.616,A -85,B 0,C 180,E1 -28830.631,E2 -28830.631} C_VEL
LIN {X 0,Y 66.93,Z 565.587,A -85,B 0,C 180,E1 -28835.275,E2 -28835.275} C_VEL
LIN {X 0,Y 67.015,Z 567.518,A -85,B 0,C 180,E1 -28836.147,E2 -28836.147} C_VEL
LIN {X 0,Y 65.344,Z 579.432,A -85,B 0,C 180,E1 -28841.161,E2 -28841.161} C_VEL
LIN {X 0,Y 63.669,Z 591.022,A -85,B 0,C 180,E1 -28847.461,E2 -28847.461} C_VEL
LIN {X 0,Y 62.07,Z 602.543,A -85,B 0,C 180,E1 -28855.52,E2 -28855.52} C_VEL
LIN {X 0,Y 61.298,Z 610.794,A -85,B 0,C 180,E1 -28862.703,E2 -28862.703} C_VEL
LIN {X 0,Y 60.867,Z 616.458,A -85,B 0,C 180,E1 -28868.516,E2 -28868.516} C_VEL
LIN {X 0,Y 59.693,Z 623.844,A -85,B 0,C 180,E1 -28878.111,E2 -28878.111} C_VEL
LIN {X 0,Y 60.05,Z 629.168,A -85,B 0,C 180,E1 -28886.646,E2 -28886.646} C_VEL
LIN {X 0,Y 60.853,Z 632.578,A -85,B 0,C 180,E1 -28893.311,E2 -28893.311} C_VEL
LIN {X 0,Y 59.741,Z 635.592,A -85,B 0,C 180,E1 -28903.609,E2 -28903.609} C_VEL
LIN {X 0,Y 61.427,Z 638.396,A -85,B 0,C 180,E1 -28917.237,E2 -28917.237} C_VEL
LIN {X 0,Y 66.637,Z 640.007,A -85,B 0,C 180,E1 -28929.258,E2 -28929.258} C_VEL
LIN {X 0,Y 74.628,Z 640.522,A -85,B 0,C 180,E1 -28938.886,E2 -28938.886} C_VEL
LIN {X 0,Y 84.488,Z 639.924,A -85,B 0,C 180,E1 -28946.289,E2 -28946.289} C_VEL
LIN {X 0,Y 95.407,Z 638.168,A -85,B 0,C 180,E1 -28952.126,E2 -28952.126} C_VEL
LIN {X 0,Y 106.915,Z 635.268,A -85,B 0,C 180,E1 -28956.97,E2 -28956.97} C_VEL
LIN {X 0,Y 109.26,Z 634.447,A -85,B 0,C 180,E1 -28958.323,E2 -28958.323} C_VEL
LIN {X 0,Y 96.918,Z 635.137,A -85,B 0,C 180,E1 -28963.14,E2 -28963.14} C_VEL
LIN {X 0,Y 85.896,Z 634.363,A -85,B 0,C 180,E1 -28969.068,E2 -28969.068} C_VEL
LIN {X 0,Y 77.583,Z 632.629,A -85,B 0,C 180,E1 -28975.183,E2 -28975.183} C_VEL
LIN {X 0,Y 70.359,Z 629.863,A -85,B 0,C 180,E1 -28982.698,E2 -28982.698} C_VEL
LIN {X 0,Y 64.138,Z 625.629,A -85,B 0,C 180,E1 -28992.661,E2 -28992.661} C_VEL
LIN {X 0,Y 60.011,Z 619.607,A -85,B 0,C 180,E1 -29004.895,E2 -29004.895} C_VEL
LIN {X 0,Y 58.738,Z 612.799,A -85,B 0,C 180,E1 -29016.747,E2 -29016.747} C_VEL
LIN {X 0,Y 59.56,Z 605.24,A -85,B 0,C 180,E1 -29027.521,E2 -29027.521} C_VEL
LIN {X 0,Y 62.438,Z 595.492,A -85,B 0,C 180,E1 -29038.158,E2 -29038.158} C_VEL
LIN {X 0,Y 66.177,Z 585.012,A -85,B 0,C 180,E1 -29046.617,E2 -29046.617} C_VEL
LIN {X 0,Y 69.324,Z 576.773,A -85,B 0,C 180,E1 -29051.642,E2 -29051.642} C_VEL
LIN {X 0,Y 69.456,Z 575.665,A -85,B 0,C 180,E1 -29052.328,E2 -29052.328} C_VEL
LIN {X 0,Y 67.477,Z 565.41,A -85,B 0,C 180,E1 -29059.497,E2 -29059.497} C_VEL
LIN {X 0,Y 65.305,Z 556.623,A -85,B 0,C 180,E1 -29065.524,E2 -29065.524} C_VEL
LIN {X 0,Y 62.471,Z 548.17,A -85,B 0,C 180,E1 -29071.611,E2 -29071.611} C_VEL
LIN {X 0,Y 59.214,Z 542.753,A -85,B 0,C 180,E1 -29076.816,E2 -29076.816} C_VEL
LIN {X 0,Y 58.732,Z 541.16,A -85,B 0,C 180,E1 -29078.168,E2 -29078.168} C_VEL
LIN {X 0,Y 58.513,Z 541.189,A -85,B 0,C 180,E1 -29086.072,E2 -29086.072} C_VEL
LIN {X 0,Y 58.131,Z 541.243,A -85,B 0,C 180,E1 -29098.92,E2 -29098.92} C_VEL
LIN {X 0,Y 58.022,Z 541.256,A -85,B 0,C 180,E1 -29107.274,E2 -29107.274} C_VEL
LIN {X 0,Y 58.003,Z 541.255,A -85,B 0,C 180,E1 -29107.623,E2 -29107.623} C_VEL
LIN {X 0,Y 57.515,Z 541.314,A -85,B 0,C 180,E1 -29111.492,E2 -29111.492} C_VEL
LIN {X 0,Y 56.012,Z 541.508,A -85,B 0,C 180,E1 -29117.28,E2 -29117.28} C_VEL
LIN {X 0,Y 52.843,Z 541.9,A -85,B 0,C 180,E1 -29127.375,E2 -29127.375} C_VEL
LIN {X 0,Y 51.204,Z 542.103,A -85,B 0,C 180,E1 -29136.262,E2 -29136.262} C_VEL
LIN {X 0,Y 51.178,Z 542.098,A -85,B 0,C 180,E1 -29140.86,E2 -29140.86} C_VEL
LIN {X 0,Y 51.458,Z 542.074,A -85,B 0,C 180,E1 -29144.146,E2 -29144.146} C_VEL
LIN {X 0,Y 51.675,Z 542.048,A -85,B 0,C 180,E1 -29152.181,E2 -29152.181} C_VEL
LIN {X 0,Y 52.255,Z 541.976,A -85,B 0,C 180,E1 -29159.998,E2 -29159.998} C_VEL
LIN {X 0,Y 51.55,Z 542.054,A -85,B 0,C 180,E1 -29173.048,E2 -29173.048} C_VEL
LIN {X 0,Y 52.676,Z 545.251,A -85,B 0,C 180,E1 -29175.97,E2 -29175.97} C_VEL
LIN {X 0,Y 53.843,Z 547.034,A -85,B 0,C 180,E1 -29178.057,E2 -29178.057} C_VEL
LIN {X 0,Y 55.634,Z 550.332,A -85,B 0,C 180,E1 -29181.294,E2 -29181.294} C_VEL
LIN {X 0,Y 57.054,Z 552.876,A -85,B 0,C 180,E1 -29183.598,E2 -29183.598} C_VEL
LIN {X 0,Y 59.036,Z 560.087,A -85,B 0,C 180,E1 -29188.435,E2 -29188.435} C_VEL
LIN {X 0,Y 60.595,Z 567.714,A -85,B 0,C 180,E1 -29193.083,E2 -29193.083} C_VEL
LIN {X 0,Y 58.699,Z 579.912,A -85,B 0,C 180,E1 -29198.901,E2 -29198.901} C_VEL
LIN {X 0,Y 56.723,Z 591.491,A -85,B 0,C 180,E1 -29206.091,E2 -29206.091} C_VEL
LIN {X 0,Y 55.009,Z 602.534,A -85,B 0,C 180,E1 -29214.907,E2 -29214.907} C_VEL
LIN {X 0,Y 54.16,Z 611.576,A -85,B 0,C 180,E1 -29224.06,E2 -29224.06} C_VEL
LIN {X 0,Y 53.785,Z 615.625,A -85,B 0,C 180,E1 -29228.941,E2 -29228.941} C_VEL
LIN {X 0,Y 52.808,Z 623.277,A -85,B 0,C 180,E1 -29240.425,E2 -29240.425} C_VEL
LIN {X 0,Y 53.563,Z 628.477,A -85,B 0,C 180,E1 -29250.001,E2 -29250.001} C_VEL
LIN {X 0,Y 54.048,Z 630.233,A -85,B 0,C 180,E1 -29253.729,E2 -29253.729} C_VEL
LIN {X 0,Y 53.12,Z 633.448,A -85,B 0,C 180,E1 -29265.345,E2 -29265.345} C_VEL
LIN {X 0,Y 55.361,Z 636.479,A -85,B 0,C 180,E1 -29280.518,E2 -29280.518} C_VEL
LIN {X 0,Y 61.371,Z 638.361,A -85,B 0,C 180,E1 -29293.402,E2 -29293.402} C_VEL
LIN {X 0,Y 70.205,Z 639.136,A -85,B 0,C 180,E1 -29303.214,E2 -29303.214} C_VEL
LIN {X 0,Y 80.755,Z 638.81,A -85,B 0,C 180,E1 -29310.493,E2 -29310.493} C_VEL
LIN {X 0,Y 92.274,Z 637.349,A -85,B 0,C 180,E1 -29316.063,E2 -29316.063} C_VEL
LIN {X 0,Y 95.923,Z 636.404,A -85,B 0,C 180,E1 -29318.511,E2 -29318.511} C_VEL
LIN {X 0,Y 88.769,Z 636.138,A -85,B 0,C 180,E1 -29321.538,E2 -29321.538} C_VEL
LIN {X 0,Y 79.511,Z 634.962,A -85,B 0,C 180,E1 -29326.486,E2 -29326.486} C_VEL
LIN {X 0,Y 69.34,Z 632.298,A -85,B 0,C 180,E1 -29334.184,E2 -29334.184} C_VEL
LIN {X 0,Y 61.354,Z 628.452,A -85,B 0,C 180,E1 -29343.539,E2 -29343.539} C_VEL
LIN {X 0,Y 55.627,Z 623.535,A -85,B 0,C 180,E1 -29354.638,E2 -29354.638} C_VEL
LIN {X 0,Y 52.288,Z 617.076,A -85,B 0,C 180,E1 -29368.065,E2 -29368.065} C_VEL
LIN {X 0,Y 51.69,Z 609.938,A -85,B 0,C 180,E1 -29380.729,E2 -29380.729} C_VEL
LIN {X 0,Y 53.283,Z 601.827,A -85,B 0,C 180,E1 -29392.319,E2 -29392.319} C_VEL
LIN {X 0,Y 56.509,Z 592.584,A -85,B 0,C 180,E1 -29402.397,E2 -29402.397} C_VEL
LIN {X 0,Y 60.571,Z 582.301,A -85,B 0,C 180,E1 -29410.684,E2 -29410.684} C_VEL
LIN {X 0,Y 62.486,Z 577.593,A -85,B 0,C 180,E1 -29413.668,E2 -29413.668} C_VEL
LIN {X 0,Y 62.397,Z 575.366,A -85,B 0,C 180,E1 -29415.319,E2 -29415.319} C_VEL
LIN {X 0,Y 60.719,Z 566.057,A -85,B 0,C 180,E1 -29422.555,E2 -29422.555} C_VEL
LIN {X 0,Y 58.971,Z 558.481,A -85,B 0,C 180,E1 -29428.464,E2 -29428.464} C_VEL
LIN {X 0,Y 57.102,Z 552.417,A -85,B 0,C 180,E1 -29433.531,E2 -29433.531} C_VEL
LIN {X 0,Y 54.258,Z 547.194,A -85,B 0,C 180,E1 -29439.317,E2 -29439.317} C_VEL
LIN {X 0,Y 51.675,Z 542.896,A -85,B 0,C 180,E1 -29444.773,E2 -29444.773} C_VEL
LIN {X 0,Y 51.46,Z 542.067,A -85,B 0,C 180,E1 -29445.85,E2 -29445.85} C_VEL
LIN {X 0,Y 51.014,Z 542.123,A -85,B 0,C 180,E1 -29454.411,E2 -29454.411} C_VEL
LIN {X 0,Y 50.987,Z 542.124,A -85,B 0,C 180,E1 -29464.2,E2 -29464.2} C_VEL
LIN {X 0,Y 50.977,Z 542.126,A -85,B 0,C 180,E1 -29473.576,E2 -29473.576} C_VEL
LIN {X 0,Y 51.03,Z 542.129,A -85,B 0,C 180,E1 -29485.724,E2 -29485.724} C_VEL
LIN {X 0,Y 51.024,Z 542.128,A -85,B 0,C 180,E1 -29495.59,E2 -29495.59} C_VEL
LIN {X 0,Y 51.178,Z 542.098,A -85,B 0,C 180,E1 -29500.86,E2 -29500.86} C_VEL
LIN {X 0,Y 50.807,Z 542.155,A -85,B 0,C 180,E1 -29504.644,E2 -29504.644} C_VEL
LIN {X 0,Y 48.982,Z 542.38,A -85,B 0,C 180,E1 -29509.831,E2 -29509.831} C_VEL
LIN {X 0,Y 45.435,Z 543.324,A -85,B 0,C 180,E1 -29519.894,E2 -29519.894} C_VEL
LIN {X 0,Y 45.238,Z 544.698,A -85,B 0,C 180,E1 -29524.127,E2 -29524.127} C_VEL
LIN {X 0,Y 45.438,Z 545.259,A -85,B 0,C 180,E1 -29525.121,E2 -29525.121} C_VEL
LIN {X 0,Y 47.541,Z 548.193,A -85,B 0,C 180,E1 -29530.643,E2 -29530.643} C_VEL
LIN {X 0,Y 51.779,Z 556.891,A -85,B 0,C 180,E1 -29540.871,E2 -29540.871} C_VEL
LIN {X 0,Y 53.663,Z 565.355,A -85,B 0,C 180,E1 -29547.28,E2 -29547.28} C_VEL
LIN {X 0,Y 54.297,Z 569.348,A -85,B 0,C 180,E1 -29550.102,E2 -29550.102} C_VEL
LIN {X 0,Y 51.835,Z 582.034,A -85,B 0,C 180,E1 -29557.199,E2 -29557.199} C_VEL
LIN {X 0,Y 49.5,Z 593.56,A -85,B 0,C 180,E1 -29565.694,E2 -29565.694} C_VEL
LIN {X 0,Y 47.804,Z 603.479,A -85,B 0,C 180,E1 -29575.272,E2 -29575.272} C_VEL
LIN {X 0,Y 47.033,Z 612.125,A -85,B 0,C 180,E1 -29585.794,E2 -29585.794} C_VEL
LIN {X 0,Y 46.381,Z 616.552,A -85,B 0,C 180,E1 -29592.36,E2 -29592.36} C_VEL
LIN {X 0,Y 46.19,Z 623.834,A -85,B 0,C 180,E1 -29605.638,E2 -29605.638} C_VEL
LIN {X 0,Y 47.211,Z 627.745,A -85,B 0,C 180,E1 -29614.27,E2 -29614.27} C_VEL
LIN {X 0,Y 46.585,Z 630.143,A -85,B 0,C 180,E1 -29623.08,E2 -29623.08} C_VEL
LIN {X 0,Y 47.826,Z 633.305,A -85,B 0,C 180,E1 -29638.155,E2 -29638.155} C_VEL
LIN {X 0,Y 52.596,Z 635.657,A -85,B 0,C 180,E1 -29651.923,E2 -29651.923} C_VEL
LIN {X 0,Y 61.087,Z 637.221,A -85,B 0,C 180,E1 -29663.645,E2 -29663.645} C_VEL
LIN {X 0,Y 71.754,Z 637.745,A -85,B 0,C 180,E1 -29671.828,E2 -29671.828} C_VEL
LIN {X 0,Y 83.49,Z 637.137,A -85,B 0,C 180,E1 -29677.815,E2 -29677.815} C_VEL
LIN {X 0,Y 83.125,Z 636.984,A -85,B 0,C 180,E1 -29678.441,E2 -29678.441} C_VEL
LIN {X 0,Y 73.322,Z 635.353,A -85,B 0,C 180,E1 -29683.44,E2 -29683.44} C_VEL
LIN {X 0,Y 64.229,Z 632.718,A -85,B 0,C 180,E1 -29690.003,E2 -29690.003} C_VEL
LIN {X 0,Y 55.219,Z 628.462,A -85,B 0,C 180,E1 -29700.002,E2 -29700.002} C_VEL
LIN {X 0,Y 48.563,Z 622.773,A -85,B 0,C 180,E1 -29713.102,E2 -29713.102} C_VEL
LIN {X 0,Y 45.169,Z 616.103,A -85,B 0,C 180,E1 -29727.828,E2 -29727.828} C_VEL
LIN {X 0,Y 44.698,Z 608.884,A -85,B 0,C 180,E1 -29741.935,E2 -29741.935} C_VEL
LIN {X 0,Y 46.394,Z 601.187,A -85,B 0,C 180,E1 -29754.089,E2 -29754.089} C_VEL
LIN {X 0,Y 49.872,Z 592.01,A -85,B 0,C 180,E1 -29764.989,E2 -29764.989} C_VEL
LIN {X 0,Y 54.444,Z 581.166,A -85,B 0,C 180,E1 -29774.135,E2 -29774.135} C_VEL
LIN {X 0,Y 55.846,Z 577.877,A -85,B 0,C 180,E1 -29776.351,E2 -29776.351} C_VEL
LIN {X 0,Y 54.574,Z 569.503,A -85,B 0,C 180,E1 -29783.859,E2 -29783.859} C_VEL
LIN {X 0,Y 52.946,Z 561.107,A -85,B 0,C 180,E1 -29791.427,E2 -29791.427} C_VEL
LIN {X 0,Y 51.457,Z 555.787,A -85,B 0,C 180,E1 -29796.676,E2 -29796.676} C_VEL
LIN {X 0,Y 47.367,Z 548.196,A -85,B 0,C 180,E1 -29807.261,E2 -29807.261} C_VEL
LIN {X 0,Y 45.453,Z 546.478,A -85,B 0,C 180,E1 -29811.909,E2 -29811.909} C_VEL
LIN {X 0,Y 43.975,Z 543.803,A -85,B 0,C 180,E1 -29817.354,E2 -29817.354} C_VEL
LIN {X 0,Y 43.821,Z 543.023,A -85,B 0,C 180,E1 -29818.759,E2 -29818.759} C_VEL
LIN {X 0,Y 43.786,Z 543.029,A -85,B 0,C 180,E1 -29829.943,E2 -29829.943} C_VEL
LIN {X 0,Y 43.841,Z 543.016,A -85,B 0,C 180,E1 -29843.275,E2 -29843.275} C_VEL
LIN {X 0,Y 43.843,Z 543.015,A -85,B 0,C 180,E1 -29851.253,E2 -29851.253} C_VEL
LIN {X 0,Y 44.229,Z 542.976,A -85,B 0,C 180,E1 -29862.438,E2 -29862.438} C_VEL
LIN {X 0,Y 44.529,Z 542.938,A -85,B 0,C 180,E1 -29870.917,E2 -29870.917} C_VEL
LIN {X 0,Y 45.129,Z 542.864,A -85,B 0,C 180,E1 -29879.998,E2 -29879.998} C_VEL
LIN {X 0,Y 44.904,Z 542.978,A -85,B 0,C 180,E1 -29882.521,E2 -29882.521} C_VEL
LIN {X 0,Y 45.438,Z 545.259,A -85,B 0,C 180,E1 -29885.121,E2 -29885.121} C_VEL
LIN {X 0,Y 46.259,Z 548.052,A -85,B 0,C 180,E1 -29888.45,E2 -29888.45} C_VEL
LIN {X 0,Y 46.662,Z 553.627,A -85,B 0,C 180,E1 -29892.862,E2 -29892.862} C_VEL
LIN {X 0,Y 46.928,Z 562.978,A -85,B 0,C 180,E1 -29899.709,E2 -29899.709} C_VEL
LIN {X 0,Y 48.066,Z 571.136,A -85,B 0,C 180,E1 -29906.717,E2 -29906.717} C_VEL
LIN {X 0,Y 44.989,Z 583.839,A -85,B 0,C 180,E1 -29914.903,E2 -29914.903} C_VEL
LIN {X 0,Y 42.5,Z 594.258,A -85,B 0,C 180,E1 -29924.071,E2 -29924.071} C_VEL
LIN {X 0,Y 40.595,Z 604.312,A -85,B 0,C 180,E1 -29935.762,E2 -29935.762} C_VEL
LIN {X 0,Y 39.953,Z 611.901,A -85,B 0,C 180,E1 -29946.977,E2 -29946.977} C_VEL
LIN {X 0,Y 39.069,Z 618.53,A -85,B 0,C 180,E1 -29959.638,E2 -29959.638} C_VEL
LIN {X 0,Y 40,Z 624.118,A -85,B 0,C 180,E1 -29972.519,E2 -29972.519} C_VEL
LIN {X 0,Y 40.362,Z 625.109,A -85,B 0,C 180,E1 -29974.996,E2 -29974.996} C_VEL
LIN {X 0,Y 40.273,Z 626.544,A -85,B 0,C 180,E1 -29980.052,E2 -29980.052} C_VEL
LIN {X 0,Y 41.471,Z 630.747,A -85,B 0,C 180,E1 -30000.559,E2 -30000.559} C_VEL
LIN {X 0,Y 47.676,Z 633.674,A -85,B 0,C 180,E1 -30017.483,E2 -30017.483} C_VEL
LIN {X 0,Y 57.239,Z 635.524,A -85,B 0,C 180,E1 -30029.261,E2 -30029.261} C_VEL
LIN {X 0,Y 68.711,Z 636.319,A -85,B 0,C 180,E1 -30037.009,E2 -30037.009} C_VEL
LIN {X 0,Y 69.257,Z 636.014,A -85,B 0,C 180,E1 -30038.8,E2 -30038.8} C_VEL
LIN {X 0,Y 57.828,Z 632.444,A -85,B 0,C 180,E1 -30046.478,E2 -30046.478} C_VEL
LIN {X 0,Y 49.34,Z 628.289,A -85,B 0,C 180,E1 -30055.636,E2 -30055.636} C_VEL
LIN {X 0,Y 42.042,Z 622.396,A -85,B 0,C 180,E1 -30069.626,E2 -30069.626} C_VEL
LIN {X 0,Y 38.486,Z 616.453,A -85,B 0,C 180,E1 -30084.064,E2 -30084.064} C_VEL
LIN {X 0,Y 37.59,Z 608.639,A -85,B 0,C 180,E1 -30101.592,E2 -30101.592} C_VEL
LIN {X 0,Y 39.955,Z 599.254,A -85,B 0,C 180,E1 -30118.148,E2 -30118.148} C_VEL
LIN {X 0,Y 43.973,Z 589.887,A -85,B 0,C 180,E1 -30129.889,E2 -30129.889} C_VEL
LIN {X 0,Y 48.647,Z 579.854,A -85,B 0,C 180,E1 -30138.541,E2 -30138.541} C_VEL
LIN {X 0,Y 49.043,Z 578.424,A -85,B 0,C 180,E1 -30139.68,E2 -30139.68} C_VEL
LIN {X 0,Y 48.379,Z 572.465,A -85,B 0,C 180,E1 -30145.834,E2 -30145.834} C_VEL
LIN {X 0,Y 47.165,Z 564.438,A -85,B 0,C 180,E1 -30154.151,E2 -30154.151} C_VEL
LIN {X 0,Y 46.278,Z 560.37,A -85,B 0,C 180,E1 -30158.734,E2 -30158.734} C_VEL
LIN {X 0,Y 43.312,Z 554.086,A -85,B 0,C 180,E1 -30168.936,E2 -30168.936} C_VEL
LIN {X 0,Y 41.039,Z 551.116,A -85,B 0,C 180,E1 -30176.804,E2 -30176.804} C_VEL
LIN {X 0,Y 40.116,Z 549.14,A -85,B 0,C 180,E1 -30181.705,E2 -30181.705} C_VEL
LIN {X 0,Y 37.554,Z 546.565,A -85,B 0,C 180,E1 -30198.466,E2 -30198.466} C_VEL
LIN {X 0,Y 37.251,Z 545.85,A -85,B 0,C 180,E1 -30205.525,E2 -30205.525} C_VEL
LIN {X 0,Y 38.05,Z 546.452,A -85,B 0,C 180,E1 -30223.009,E2 -30223.009} C_VEL
LIN {X 0,Y 40.124,Z 548.363,A -85,B 0,C 180,E1 -30234.973,E2 -30234.973} C_VEL
LIN {X 0,Y 41.406,Z 549.698,A -85,B 0,C 180,E1 -30239.997,E2 -30239.997} C_VEL
LIN {X 0,Y 42.272,Z 551.915,A -85,B 0,C 180,E1 -30244.041,E2 -30244.041} C_VEL
LIN {X 0,Y 43.171,Z 553.136,A -85,B 0,C 180,E1 -30246.811,E2 -30246.811} C_VEL
LIN {X 0,Y 45.036,Z 557.818,A -85,B 0,C 180,E1 -30253.535,E2 -30253.535} C_VEL
LIN {X 0,Y 46.472,Z 560.78,A -85,B 0,C 180,E1 -30257.603,E2 -30257.603} C_VEL
LIN {X 0,Y 46.928,Z 562.978,A -85,B 0,C 180,E1 -30259.709,E2 -30259.709} C_VEL
LIN {X 0,Y 46.799,Z 565.857,A -85,B 0,C 180,E1 -30261.667,E2 -30261.667} C_VEL
LIN {X 0,Y 45.349,Z 570.046,A -85,B 0,C 180,E1 -30263.424,E2 -30263.424} C_VEL
LIN {X 0,Y 40.186,Z 579.384,A -85,B 0,C 180,E1 -30266.963,E2 -30266.963} C_VEL
LIN {X 0,Y 39.314,Z 581.708,A -85,B 0,C 180,E1 -30268.658,E2 -30268.658} C_VEL
LIN {X 0,Y 36.188,Z 592.41,A -85,B 0,C 180,E1 -30279.031,E2 -30279.031} C_VEL
LIN {X 0,Y 33.699,Z 602.99,A -85,B 0,C 180,E1 -30293.347,E2 -30293.347} C_VEL
LIN {X 0,Y 32.883,Z 611.196,A -85,B 0,C 180,E1 -30308.038,E2 -30308.038} C_VEL
LIN {X 0,Y 32.513,Z 619.07,A -85,B 0,C 180,E1 -30326.904,E2 -30326.904} C_VEL
LIN {X 0,Y 33.497,Z 622.338,A -85,B 0,C 180,E1 -30336.023,E2 -30336.023} C_VEL
LIN {X 0,Y 33.719,Z 623.984,A -85,B 0,C 180,E1 -30342.032,E2 -30342.032} C_VEL
LIN {X 0,Y 35.787,Z 628.406,A -85,B 0,C 180,E1 -30366.098,E2 -30366.098} C_VEL
LIN {X 0,Y 43.32,Z 631.615,A -85,B 0,C 180,E1 -30384.214,E2 -30384.214} C_VEL
LIN {X 0,Y 54.03,Z 633.705,A -85,B 0,C 180,E1 -30395.583,E2 -30395.583} C_VEL
LIN {X 0,Y 56.973,Z 633.949,A -85,B 0,C 180,E1 -30398.282,E2 -30398.282} C_VEL
LIN {X 0,Y 46.525,Z 629.519,A -85,B 0,C 180,E1 -30406.906,E2 -30406.906} C_VEL
LIN {X 0,Y 37.753,Z 623.762,A -85,B 0,C 180,E1 -30420.003,E2 -30420.003} C_VEL
LIN {X 0,Y 32.054,Z 616.812,A -85,B 0,C 180,E1 -30438.489,E2 -30438.489} C_VEL
LIN {X 0,Y 30.455,Z 608.988,A -85,B 0,C 180,E1 -30459.396,E2 -30459.396} C_VEL
LIN {X 0,Y 32.722,Z 599.734,A -85,B 0,C 180,E1 -30479.225,E2 -30479.225} C_VEL
LIN {X 0,Y 36.874,Z 590.799,A -85,B 0,C 180,E1 -30492.37,E2 -30492.37} C_VEL
LIN {X 0,Y 42.48,Z 579.641,A -85,B 0,C 180,E1 -30503.075,E2 -30503.075} C_VEL
LIN {X 0,Y 41.921,Z 572.189,A -85,B 0,C 180,E1 -30512.065,E2 -30512.065} C_VEL
LIN {X 0,Y 41.207,Z 566.008,A -85,B 0,C 180,E1 -30519.819,E2 -30519.819} C_VEL
LIN {X 0,Y 40.928,Z 564.363,A -85,B 0,C 180,E1 -30522.083,E2 -30522.083} C_VEL
LIN {X 0,Y 39.076,Z 559.688,A -85,B 0,C 180,E1 -30531.081,E2 -30531.081} C_VEL
LIN {X 0,Y 36.438,Z 555.063,A -85,B 0,C 180,E1 -30545.353,E2 -30545.353} C_VEL
LIN {X 0,Y 34.788,Z 552.719,A -85,B 0,C 180,E1 -30563.909,E2 -30563.909} C_VEL
LIN {X 0,Y 34.978,Z 552.729,A -85,B 0,C 180,E1 -30576.302,E2 -30576.302} C_VEL
LIN {X 0,Y 36.326,Z 554.045,A -85,B 0,C 180,E1 -30588.842,E2 -30588.842} C_VEL
LIN {X 0,Y 37.367,Z 554.991,A -85,B 0,C 180,E1 -30594.601,E2 -30594.601} C_VEL
LIN {X 0,Y 37.86,Z 555.816,A -85,B 0,C 180,E1 -30597.337,E2 -30597.337} C_VEL
LIN {X 0,Y 39.186,Z 558.926,A -85,B 0,C 180,E1 -30604.36,E2 -30604.36} C_VEL
LIN {X 0,Y 41.416,Z 565.452,A -85,B 0,C 180,E1 -30614.744,E2 -30614.744} C_VEL
LIN {X 0,Y 41.967,Z 572.388,A -85,B 0,C 180,E1 -30621.943,E2 -30621.943} C_VEL
LIN {X 0,Y 39.314,Z 581.708,A -85,B 0,C 180,E1 -30628.658,E2 -30628.658} C_VEL
LIN {X 0,Y 37.372,Z 586.637,A -85,B 0,C 180,E1 -30632.626,E2 -30632.626} C_VEL
LIN {X 0,Y 34.572,Z 591.299,A -85,B 0,C 180,E1 -30636.52,E2 -30636.52} C_VEL
LIN {X 0,Y 27.695,Z 601.353,A -85,B 0,C 180,E1 -30649.269,E2 -30649.269} C_VEL
LIN {X 0,Y 26.187,Z 605.507,A -85,B 0,C 180,E1 -30657.737,E2 -30657.737} C_VEL
LIN {X 0,Y 25.814,Z 610.656,A -85,B 0,C 180,E1 -30670.105,E2 -30670.105} C_VEL
LIN {X 0,Y 26.204,Z 618.332,A -85,B 0,C 180,E1 -30693.847,E2 -30693.847} C_VEL
LIN {X 0,Y 26.695,Z 619.447,A -85,B 0,C 180,E1 -30697.566,E2 -30697.566} C_VEL
LIN {X 0,Y 27.292,Z 621.274,A -85,B 0,C 180,E1 -30704.925,E2 -30704.925} C_VEL
LIN {X 0,Y 30.604,Z 625.948,A -85,B 0,C 180,E1 -30733.549,E2 -30733.549} C_VEL
LIN {X 0,Y 39.712,Z 629.403,A -85,B 0,C 180,E1 -30752.24,E2 -30752.24} C_VEL
LIN {X 0,Y 43.87,Z 630.193,A -85,B 0,C 180,E1 -30758.223,E2 -30758.223} C_VEL
LIN {X 0,Y 33.233,Z 624.061,A -85,B 0,C 180,E1 -30770.877,E2 -30770.877} C_VEL
LIN {X 0,Y 25.666,Z 616.392,A -85,B 0,C 180,E1 -30792.322,E2 -30792.322} C_VEL
LIN {X 0,Y 23.461,Z 607.392,A -85,B 0,C 180,E1 -30821.651,E2 -30821.651} C_VEL
LIN {X 0,Y 26.263,Z 598.465,A -85,B 0,C 180,E1 -30844.586,E2 -30844.586} C_VEL
LIN {X 0,Y 31.535,Z 588.565,A -85,B 0,C 180,E1 -30860.16,E2 -30860.16} C_VEL
LIN {X 0,Y 36.077,Z 580.237,A -85,B 0,C 180,E1 -30868.451,E2 -30868.451} C_VEL
LIN {X 0,Y 35.968,Z 573.392,A -85,B 0,C 180,E1 -30878.425,E2 -30878.425} C_VEL
LIN {X 0,Y 35.78,Z 568.803,A -85,B 0,C 180,E1 -30885.457,E2 -30885.457} C_VEL
LIN {X 0,Y 34.644,Z 564.957,A -85,B 0,C 180,E1 -30893.935,E2 -30893.935} C_VEL
LIN {X 0,Y 33.374,Z 562.477,A -85,B 0,C 180,E1 -30902.607,E2 -30902.607} C_VEL
LIN {X 0,Y 32.664,Z 560.861,A -85,B 0,C 180,E1 -30910.2,E2 -30910.2} C_VEL
LIN {X 0,Y 32.053,Z 559.883,A -85,B 0,C 180,E1 -30918.863,E2 -30918.863} C_VEL
LIN {X 0,Y 32.073,Z 559.254,A -85,B 0,C 180,E1 -30934.004,E2 -30934.004} C_VEL
LIN {X 0,Y 33.306,Z 560.422,A -85,B 0,C 180,E1 -30947.815,E2 -30947.815} C_VEL
LIN {X 0,Y 34.16,Z 561.596,A -85,B 0,C 180,E1 -30954.092,E2 -30954.092} C_VEL
LIN {X 0,Y 35.181,Z 565.145,A -85,B 0,C 180,E1 -30962.803,E2 -30962.803} C_VEL
LIN {X 0,Y 35.964,Z 568.544,A -85,B 0,C 180,E1 -30969.119,E2 -30969.119} C_VEL
LIN {X 0,Y 36.185,Z 573.277,A -85,B 0,C 180,E1 -30975.338,E2 -30975.338} C_VEL
LIN {X 0,Y 35.707,Z 575.387,A -85,B 0,C 180,E1 -30977.163,E2 -30977.163} C_VEL
LIN {X 0,Y 31.644,Z 586.662,A -85,B 0,C 180,E1 -30987.333,E2 -30987.333} C_VEL
LIN {X 0,Y 28.077,Z 597.021,A -85,B 0,C 180,E1 -31001.332,E2 -31001.332} C_VEL
LIN {X 0,Y 26.187,Z 605.507,A -85,B 0,C 180,E1 -31017.737,E2 -31017.737} C_VEL
LIN {X 0,Y 25.122,Z 608.083,A -85,B 0,C 180,E1 -31023.917,E2 -31023.917} C_VEL
LIN {X 0,Y 23.284,Z 610.24,A -85,B 0,C 180,E1 -31030.588,E2 -31030.588} C_VEL
LIN {X 0,Y 19.662,Z 614.603,A -85,B 0,C 180,E1 -31051.384,E2 -31051.384} C_VEL
LIN {X 0,Y 20.019,Z 616.653,A -85,B 0,C 180,E1 -31061.508,E2 -31061.508} C_VEL
LIN {X 0,Y 20.995,Z 618.421,A -85,B 0,C 180,E1 -31069.56,E2 -31069.56} C_VEL
LIN {X 0,Y 26.157,Z 623.41,A -85,B 0,C 180,E1 -31103.717,E2 -31103.717} C_VEL
LIN {X 0,Y 31.194,Z 625.405,A -85,B 0,C 180,E1 -31114.32,E2 -31114.32} C_VEL
LIN {X 0,Y 30.132,Z 624.389,A -85,B 0,C 180,E1 -31118.906,E2 -31118.906} C_VEL
LIN {X 0,Y 20.342,Z 616.582,A -85,B 0,C 180,E1 -31140.005,E2 -31140.005} C_VEL
LIN {X 0,Y 16.392,Z 607.963,A -85,B 0,C 180,E1 -31175.641,E2 -31175.641} C_VEL
LIN {X 0,Y 19.137,Z 598.821,A -85,B 0,C 180,E1 -31208.451,E2 -31208.451} C_VEL
LIN {X 0,Y 25.617,Z 588.295,A -85,B 0,C 180,E1 -31228.073,E2 -31228.073} C_VEL
LIN {X 0,Y 29.662,Z 581.86,A -85,B 0,C 180,E1 -31234.808,E2 -31234.808} C_VEL
LIN {X 0,Y 30.022,Z 580.802,A -85,B 0,C 180,E1 -31236.15,E2 -31236.15} C_VEL
LIN {X 0,Y 30.451,Z 575.101,A -85,B 0,C 180,E1 -31246.113,E2 -31246.113} C_VEL
LIN {X 0,Y 30.442,Z 571.915,A -85,B 0,C 180,E1 -31252.551,E2 -31252.551} C_VEL
LIN {X 0,Y 30.13,Z 570.061,A -85,B 0,C 180,E1 -31257.806,E2 -31257.806} C_VEL
LIN {X 0,Y 29.549,Z 568.571,A -85,B 0,C 180,E1 -31264.075,E2 -31264.075} C_VEL
LIN {X 0,Y 29.084,Z 566.831,A -85,B 0,C 180,E1 -31273.531,E2 -31273.531} C_VEL
LIN {X 0,Y 28.828,Z 565.75,A -85,B 0,C 180,E1 -31290.814,E2 -31290.814} C_VEL
LIN {X 0,Y 29.908,Z 566.639,A -85,B 0,C 180,E1 -31306.405,E2 -31306.405} C_VEL
LIN {X 0,Y 30.187,Z 567.068,A -85,B 0,C 180,E1 -31309.104,E2 -31309.104} C_VEL
LIN {X 0,Y 30.669,Z 569.646,A -85,B 0,C 180,E1 -31317.331,E2 -31317.331} C_VEL
LIN {X 0,Y 30.948,Z 573.135,A -85,B 0,C 180,E1 -31324.911,E2 -31324.911} C_VEL
LIN {X 0,Y 30.751,Z 575.289,A -85,B 0,C 180,E1 -31328.137,E2 -31328.137} C_VEL
LIN {X 0,Y 25.984,Z 586.219,A -85,B 0,C 180,E1 -31338.804,E2 -31338.804} C_VEL
LIN {X 0,Y 21.853,Z 595.728,A -85,B 0,C 180,E1 -31353.685,E2 -31353.685} C_VEL
LIN {X 0,Y 19.155,Z 604.847,A -85,B 0,C 180,E1 -31376.612,E2 -31376.612} C_VEL
LIN {X 0,Y 18.78,Z 609.944,A -85,B 0,C 180,E1 -31393.702,E2 -31393.702} C_VEL
LIN {X 0,Y 20.019,Z 616.653,A -85,B 0,C 180,E1 -31421.508,E2 -31421.508} C_VEL
LIN {X 0,Y 19.979,Z 617.33,A -85,B 0,C 180,E1 -31426.042,E2 -31426.042} C_VEL
LIN {X 0,Y 18.679,Z 617.538,A -85,B 0,C 180,E1 -31434.011,E2 -31434.011} C_VEL
LIN {X 0,Y 15.838,Z 616.61,A -85,B 0,C 180,E1 -31446.567,E2 -31446.567} C_VEL
LIN {X 0,Y 13.675,Z 615.353,A -85,B 0,C 180,E1 -31456.94,E2 -31456.94} C_VEL
LIN {X 0,Y 10.29,Z 612.228,A -85,B 0,C 180,E1 -31483.712,E2 -31483.712} C_VEL
LIN {X 0,Y 9.156,Z 608.496,A -85,B 0,C 180,E1 -31519.217,E2 -31519.217} C_VEL
LIN {X 0,Y 9.394,Z 605.578,A -85,B 0,C 180,E1 -31542.011,E2 -31542.011} C_VEL
LIN {X 0,Y 14.099,Z 596.395,A -85,B 0,C 180,E1 -31585.632,E2 -31585.632} C_VEL
LIN {X 0,Y 21.549,Z 586.343,A -85,B 0,C 180,E1 -31601.893,E2 -31601.893} C_VEL
LIN {X 0,Y 23.924,Z 582.997,A -85,B 0,C 180,E1 -31604.825,E2 -31604.825} C_VEL
LIN {X 0,Y 24.538,Z 581.667,A -85,B 0,C 180,E1 -31606.641,E2 -31606.641} C_VEL
LIN {X 0,Y 25.563,Z 576.885,A -85,B 0,C 180,E1 -31616.956,E2 -31616.956} C_VEL
LIN {X 0,Y 25.571,Z 574.762,A -85,B 0,C 180,E1 -31624.45,E2 -31624.45} C_VEL
LIN {X 0,Y 25.344,Z 572.866,A -85,B 0,C 180,E1 -31635.76,E2 -31635.76} C_VEL
LIN {X 0,Y 25.249,Z 572.24,A -85,B 0,C 180,E1 -31646.618,E2 -31646.618} C_VEL
LIN {X 0,Y 26.192,Z 572.659,A -85,B 0,C 180,E1 -31664.431,E2 -31664.431} C_VEL
LIN {X 0,Y 26.316,Z 573.728,A -85,B 0,C 180,E1 -31669.176,E2 -31669.176} C_VEL
LIN {X 0,Y 26.101,Z 576.478,A -85,B 0,C 180,E1 -31676.864,E2 -31676.864} C_VEL
LIN {X 0,Y 24.456,Z 579.859,A -85,B 0,C 180,E1 -31679.996,E2 -31679.996} C_VEL
LIN {X 0,Y 18.099,Z 591.164,A -85,B 0,C 180,E1 -31693.9,E2 -31693.9} C_VEL
LIN {X 0,Y 13.282,Z 600.39,A -85,B 0,C 180,E1 -31718.006,E2 -31718.006} C_VEL
LIN {X 0,Y 11.88,Z 607.679,A -85,B 0,C 180,E1 -31752.8,E2 -31752.8} C_VEL
LIN {X 0,Y 14.958,Z 615.49,A -85,B 0,C 180,E1 -31798.029,E2 -31798.029} C_VEL
LIN {X 0,Y 20.185,Z 619.539,A -85,B 0,C 180,E1 -31830.535,E2 -31830.535} C_VEL
LIN {X 0,Y 18.14,Z 617.866,A -85,B 0,C 180,E1 -31837.211,E2 -31837.211} C_VEL
LIN {X 0,Y 10.61,Z 610.351,A -85,B 0,C 180,E1 -31868.435,E2 -31868.435} C_VEL
LIN {X 0,Y 9.394,Z 605.578,A -85,B 0,C 180,E1 -31902.011,E2 -31902.011} C_VEL
LIN {X 0,Y 9.465,Z 602.947,A -85,B 0,C 180,E1 -31919.658,E2 -31919.658} C_VEL
LIN {X 0,Y 9.71,Z 598.399,A -85,B 0,C 180,E1 -31949.253,E2 -31949.253} C_VEL
LIN {X 0,Y 11.915,Z 593.528,A -85,B 0,C 180,E1 -31972.032,E2 -31972.032} C_VEL
LIN {X 0,Y 14.258,Z 590.428,A -85,B 0,C 180,E1 -31977.406,E2 -31977.406} C_VEL
LIN {X 0,Y 19.983,Z 583.238,A -85,B 0,C 180,E1 -31980.696,E2 -31980.696} C_VEL
LIN {X 0,Y 21.069,Z 580.723,A -85,B 0,C 180,E1 -31986.961,E2 -31986.961} C_VEL
LIN {X 0,Y 21.241,Z 579.763,A -85,B 0,C 180,E1 -31991.431,E2 -31991.431} C_VEL
LIN {X 0,Y 21.394,Z 578.722,A -85,B 0,C 180,E1 -31998.921,E2 -31998.921} C_VEL
LIN {X 0,Y 22.054,Z 578.593,A -85,B 0,C 180,E1 -32021.412,E2 -32021.412} C_VEL
LIN {X 0,Y 21.954,Z 579.001,A -85,B 0,C 180,E1 -32023.064,E2 -32023.064} C_VEL
LIN {X 0,Y 15.579,Z 588.599,A -85,B 0,C 180,E1 -32030.452,E2 -32030.452} C_VEL
LIN {X 0,Y 8.426,Z 598.084,A -85,B 0,C 180,E1 -32049.278,E2 -32049.278} C_VEL
LIN {X 0,Y 4.841,Z 605.259,A -85,B 0,C 180,E1 -32108.732,E2 -32108.732} C_VEL
LIN {X 0,Y 5.767,Z 608.315,A -85,B 0,C 180,E1 -32147.749,E2 -32147.749} C_VEL
LIN {X 0,Y 9.502,Z 612.183,A -85,B 0,C 180,E1 -32177.709,E2 -32177.709} C_VEL
LIN {X 0,Y 8.934,Z 611.75,A -85,B 0,C 180,E1 -32181.882,E2 -32181.882} C_VEL
LIN {X 0,Y 4.05,Z 601.666,A -85,B 0,C 180,E1 -32309.987,E2 -32309.987} C_VEL
LIN {X 0,Y 14.258,Z 590.428,A -85,B 0,C 180,E1 -32337.406,E2 -32337.406} C_VEL
LIN {X 0,Y 17.708,Z 591.754,A -85,B 0,C 180,E1 -32339.48,E2 -32339.48} C_VEL
LIN {X 0,Y 17.708,Z 600,A -85,B 0,C 180,E1 -32339.48,E2 -32339.48} C_VEL
LIN {X 0,Y 17.708,Z 600,A -85,B 0,C 180,E1 -32339.48,E2 -32339.48}

QRS_NEXT_CUT()

QRS_NEXT()
QRS_HOME()

END
